# B&R Automation Studio project Soiled_PLC (part 4)

#### pic.st - Implementation code
```iecst
(********************************************************************
 * COPYRIGHT --
 ********************************************************************
 * Program: pic
 * File: pic.st
 * Author: treamsbottom
 * Created: July 16, 2015
 ********************************************************************
 * Implementation of program pic - Pneumatic Incline
 ********************************************************************)
//V1.00.1 First Release
PROGRAM _INIT
//Configuration
mySeq						:= 23;	//Sequence number
myIO						:= 8;
myZone						:= 0;
myRelLine					:= 44;
myBuffBag					:= 0;
myBag						:= 0;
bufferSettleTime			:= 300;
myPI						:= 3;

myOutBag 					:= Line[myRelLine].LastBag;
END_PROGRAM

PROGRAM _CYCLIC
//Inputs

i_bagInIncline			:= X[myIO].X04;
i_cylinderAtBottom		:= X[myIO].X06;
i_cylinderAtTop			:= X[myIO].X05;
i_bagAtBuffer			:= X[myIO].X03;

i_bagAtBufferOut 		:= FALSE; // Any Single bag buffer out IO.
i_bufferOutOpen			:= FALSE;

o_openBuffer			:= FALSE;
o_cylinderDown			:= FALSE;

Request.PI[myPI]		:= FALSE;
RequestRel.PI[myPI]		:= FALSE;

IF (myBag = 0) THEN
//	Alarm[mySeq].Bag	:= mySeq + 10000;
ELSE
//	Alarm[mySeq].Bag	:= myBag;
END_IF;

Alarm[mySeq].Name 		:= 0;
Alarm[mySeq].Bag	:= 10017;
Alarm[mySeq].Beacon	:= TRUE;
Alarm[mySeq].Extra		:= 0;
Alarm[mySeq].Time		:= 3000;

//Setup Sequence
step := D[900 + mySeq];
//Setup Pulse contact
pls := (step <> lastStep);
lastStep := step;

//Sequence
IF (step = 0) THEN
	//Disabled
END_IF;

//Wait for at buffer
ton_10ms_SettledBuffer(IN:= i_bagAtBuffer, PT:= bufferSettleTime);
IF (step = 1) THEN
	IF NOT Std.HaltSysZone[myZone] AND i_cylinderAtTop AND NOT i_bagInIncline THEN
		IF useRequest THEN
			D[900 + mySeq] := 2;
		ELSE
			IF ton_10ms_SettledBuffer.Q THEN
				IF (myBuffBag > 0) THEN
					IF (Bag[myBuffBag].Cat > 0) AND (Bag[myBag].Cat = 0) THEN
						D[900 + mySeq] := 2;
					ELSIF (Bag[myBuffBag].Cat = 0) THEN
						Alarm[mySeq].Name := ALM_BAG_DATA_ERROR;
						Alarm[mySeq].Bag := myBuffBag;
					ELSE
						Alarm[mySeq].Name := ALM_BAG_DATA_ERROR;
					END_IF;
				ELSE
					D[900 + mySeq] := 2;
				END_IF;
			ELSIF (myBuffBag > 0) AND (Bag[myBuffBag].Cat > 0) THEN
				Alarm[mySeq].Name := ALM_BAG_NOT_SETTLED;
			END_IF;
		END_IF;
	ELSIF NOT Std.HaltSysZone[myZone] THEN
		Alarm[mySeq].Name := ALM_SWITCH_FAULT;
	END_IF;
END_IF;

//Open Buffer stop
IF (step = 2) THEN
	releaseValid := ((myBag = 0) OR ((Bag[myBag].Cat = 0) AND (Bag[myBuffBag].Cat > 0)));
	o_openBuffer	   := releaseValid AND NOT useRequest;
	Request.PI[myPI]  := releaseValid AND useRequest;
	IF (i_bagInIncline AND releaseValid) THEN
		IF (myBag > 0) THEN
			Bag[myBag] := Bag[myBuffBag]; //Clear empty buffer bag data if used
			Bag[myBuffBag] := Bag[0];
		END_IF;
		D[900 + mySeq] := 3;
	ELSIF (myBag > 0) THEN
		IF (Bag[myBag].Cat > 0) THEN
			Alarm[mySeq].Name := ALM_BAG_DATA_ERROR;
			Alarm[mySeq].Time := 0;
		ELSIF (Bag[myBuffBag].Cat = 0) THEN
			Alarm[mySeq].Name := ALM_BAG_DATA_ERROR;
			Alarm[mySeq].Bag := myBuffBag;
			Alarm[mySeq].Time := 0;
		ELSE
			Alarm[mySeq].Name  := ALM_BAG_NOT_ARRIVED;
		END_IF;
		Alarm[mySeq].Name  := ALM_BAG_NOT_ARRIVED;
	END_IF;
END_IF;

//Let bag settle at base OF incline
ton_10ms_SettledInIncline(IN:= i_bagInIncline, PT:= 300);
IF (step = 3) THEN
	o_openBuffer := NOT useRequest;
	IF  ton_10ms_SettledInIncline.Q AND NOT Std.HaltSysZone[myZone] THEN
		D[900 + mySeq] := 4;
	ELSIF NOT Std.HaltSysZone[myZone] THEN
		Alarm[mySeq].Name := ALM_BAG_NOT_SETTLED;
	END_IF;
END_IF

//Move incline down to collect first trolley
ton_10ms_CylinderDown(IN := i_cylinderAtBottom, PT:=300);
IF (step = 4) THEN
	o_openBuffer := NOT useRequest;
	o_cylinderDown := TRUE;
	IF ton_10ms_CylinderDown.Q THEN
		D[900 + mySeq] := 5;
	END_IF;
	Alarm[mySeq].Name := ALM_SWITCH_FAULT;
END_IF;

//Let cylinder move back to the top.
IF (step = 5) THEN
	o_openBuffer := NOT useRequest;
	IF i_cylinderAtTop THEN
		D[900 + mySeq] := 6;
	END_IF;
	Alarm[mySeq].Name := ALM_SWITCH_FAULT;
END_IF;

//Check for valid release..
//Check for line space.
IF (step = 6) THEN
	releaseValid := (ton_10ms_SettledInIncline.Q AND NOT i_cylinderAtBottom AND NOT i_bagAtBufferOut AND NOT i_bufferOutOpen AND ((myBag = 0) OR ((Bag[myBag].Cat > 0) AND (Bag[myOutBag].Cat = 0))));
	IF (myRelLine > 0) THEN
		IF (Line[myRelLine].Clear AND releaseValid) THEN
			C[myRelLine] := 0;
			D[900 + mySeq] := 7;
		END_IF;
		IF i_cylinderAtBottom OR NOT i_bagInIncline THEN
			Alarm[mySeq].Name := ALM_SWITCH_FAULT;
			Alarm[mySeq].Time := 0;
		ELSIF (Line[myRelLine].Clear AND i_bagAtBufferOut) THEN
			Alarm[mySeq].Name := ALM_SWITCH_FAULT;
		ELSIF (myBag > 0) AND (Bag[myBag].Cat = 0) THEN
			Alarm[mySeq].Name := ALM_BAG_DATA_ERROR;
			Alarm[mySeq].Time := 0;
		ELSIF Line[myRelLine].Clear AND (myOutBag > 0) AND (Bag[myOutBag].Cat > 0) THEN
			Alarm[mySeq].Name := ALM_BAG_DATA_ERROR;
			Alarm[mySeq].Bag := myOutBag;
			Alarm[mySeq].Time := 0;
		END_IF;
	ELSE
		RequestRel.PI[myPI] := releaseValid;
		IF EnableRel.PI[myPI] AND releaseValid THEN
			D[900 + mySeq] := 7;
		ELSIF NOT i_cylinderAtBottom OR NOT i_bagInIncline THEN
			Alarm[mySeq].Name := ALM_SWITCH_FAULT;
			Alarm[mySeq].Time := 0;
		ELSIF (myBag > 0) AND (Bag[myBag].Cat = 0) THEN
			Alarm[mySeq].Name := ALM_BAG_DATA_ERROR;
			Alarm[mySeq].Time := 0;
		ELSIF (myOutBag > 0) AND (Bag[myOutBag].Cat > 0) THEN
			Alarm[mySeq].Name := ALM_BAG_DATA_ERROR;
			Alarm[mySeq].Bag := myOutBag;
			Alarm[mySeq].Time := 0;
		END_IF;
	END_IF;
END_IF;

//Move cylinder down to get 2nd trolley.
IF (step = 7) THEN
	o_cylinderDown := TRUE;
	IF  ton_10ms_CylinderDown.Q THEN
		D[900 + mySeq] := 8;
	END_IF;
	Alarm[mySeq].Name := ALM_SWITCH_FAULT;
END_IF;

//Release bag
IF (step = 8) THEN
	releaseValid := (NOT i_bagAtBufferOut AND NOT i_bufferOutOpen AND ((myBag = 0) OR ((Bag[myBag].Cat > 0) AND (Bag[myOutBag].Cat = 0))));
	o_cylinderDown := NOT releaseValid; // Hold cylinder down if release is not valid.
	IF releaseValid THEN
		IF (myBag = 0) THEN// Not tracking.
			IF (myRelLine > 0) THEN
				IF Line[myRelLine].Trip THEN
					D[900 + mySeq] := 1;
				END_IF;
			ELSE
				IF NOT EnableRel.PI[myPI] THEN
					D[900 + mySeq] := 1;
				END_IF;
			END_IF;
			IF NOT Std.HaltSysZone[myZone] THEN
				Alarm[mySeq].Name := ALM_BAG_NOT_RELEASED;
			END_IF;
		ELSE//Use tracking
			IF (myRelLine > 0) THEN
				IF Line[myRelLine].Trip THEN
					Bag[myOutBag] := Bag[myBag];
					Bag[myBag] := Bag[0];
					D[900 + mySeq] := 1;
				END_IF;
			ELSE
				IF NOT EnableRel.PI[myPI] AND (Bag[myBag].Cat = 0) THEN // Make sure data is copied out by enabling sequence.
					D[900 + mySeq] := 1;
				ELSIF NOT EnableRel.PI[myPI] AND (Bag[myBag].Cat > 0) THEN
					Alarm[mySeq].Name := ALM_BAG_DATA_ERROR;
				END_IF;
			END_IF;
		END_IF;
	ELSIF i_bagAtBufferOut AND NOT i_bufferOutOpen THEN
		Alarm[mySeq].Name := ALM_SWITCH_FAULT;
		Alarm[mySeq].Time := 0;
	ELSIF (myBag > 0) THEN
		IF (Bag[myBag].Cat = 0) THEN
			Alarm[mySeq].Name := ALM_BAG_DATA_ERROR;
			Alarm[mySeq].Time := 0;
		ELSIF (Bag[myOutBag].Cat > 0) THEN
			Alarm[mySeq].Name := ALM_BAG_DATA_ERROR;
			Alarm[mySeq].Bag := myOutBag;
			Alarm[mySeq].Time := 0;
		END_IF;
	END_IF;
END_IF

//-----------------------------------
//PLC Outputs - adjust TO suit system
//-----------------------------------

Y[11].Y09 := o_cylinderDown;
Y[3].Y15 := o_openBuffer;

//Alarms
timerAlarm(IN := NOT pls AND (Alarm[mySeq].Name > 0),PT:= Alarm[mySeq].Time);

Alarm[mySeq].On 	:= timerAlarm.Q;
Alarm[mySeq].ET 	:= timerAlarm.ET;

END_PROGRAM
```

#### pic.var - Local variables
```iecst
(********************************************************************
 * COPYRIGHT --
 ********************************************************************
 * Program: pr
 * File: pr.var
 * Author: treamsbottom
 * Created: July 16, 2015
 ********************************************************************
 * Local variables of program pr
 ********************************************************************)
VAR
	mySeq : UINT;
	myIO : UINT;
	myZone : UINT;
	myRelLine : UINT;
	myBag : UINT;
	i_bagAtBuffer : BOOL;
	i_bagAtBufferOut : BOOL;
	i_bufferOutOpen : BOOL;
	o_openBuffer : BOOL;
	step : UINT;
	pls : BOOL;
	timerAlarm : TON_10ms;
END_VAR
VAR RETAIN
	lastStep : UINT;
END_VAR
VAR
	bufferSettleTime : UDINT;
	myOutBag : UINT;
	myBuffBag : UINT;
	myPI : UINT;
	i_bagInIncline : BOOL;
	i_cylinderAtBottom : BOOL;
	i_cylinderAtTop : BOOL;
	o_cylinderDown : BOOL;
	useRequest : BOOL;
	releaseValid : BOOL;
	ton_10ms_SettledBuffer : TON_10ms;
	ton_10ms_SettledInIncline : TON_10ms;
	ton_10ms_CylinderDown : TON_10ms;
END_VAR
```

### Program Logical/Sequences/10ms/24_cpi4 (IEC) - *Pneumatic Incline

#### pic.st
```iecst
(********************************************************************
 * COPYRIGHT --
 ********************************************************************
 * Program: pic
 * File: pic.st
 * Author: treamsbottom
 * Created: July 16, 2015
 ********************************************************************
 * Implementation of program pic - Pneumatic Incline
 ********************************************************************)
//V1.00.1 First Release
PROGRAM _INIT
//Configuration
mySeq						:= 24;	//Sequence number
myIO						:= 7;
myZone						:= 0;
myRelLine					:= 41;
myBuffBag					:= 0;
myBag						:= 0;
bufferSettleTime			:= 300;
myPI						:= 4;

myOutBag 					:= Line[myRelLine].LastBag;
END_PROGRAM

PROGRAM _CYCLIC
//Inputs

i_bagInIncline			:= X[9].X16;
i_cylinderAtBottom		:= X[10].X01;
i_cylinderAtTop			:= X[10].X02;
i_bagAtBuffer			:= X[9].X15;

i_bagAtBufferOut 		:= FALSE; // Any Single bag buffer out IO.
i_bufferOutOpen			:= FALSE;

o_openBuffer			:= FALSE;
o_cylinderDown			:= FALSE;

Request.PI[myPI]		:= FALSE;
RequestRel.PI[myPI]		:= FALSE;

IF (myBag = 0) THEN
//	Alarm[mySeq].Bag	:= mySeq + 10000;
ELSE
//	Alarm[mySeq].Bag	:= myBag;
END_IF;

Alarm[mySeq].Name 		:= 0;
Alarm[mySeq].Bag	:= 10018;
Alarm[mySeq].Beacon	:= TRUE;
Alarm[mySeq].Extra		:= 0;
Alarm[mySeq].Time		:= 3000;

//Setup Sequence
step := D[900 + mySeq];
//Setup Pulse contact
pls := (step <> lastStep);
lastStep := step;

//Sequence
IF (step = 0) THEN
	//Disabled
END_IF;

//Wait for at buffer
ton_10ms_SettledBuffer(IN:= i_bagAtBuffer, PT:= bufferSettleTime);
IF (step = 1) THEN
	IF NOT Std.HaltSysZone[myZone] AND i_cylinderAtTop AND NOT i_bagInIncline THEN
		IF useRequest THEN
			D[900 + mySeq] := 2;
		ELSE
			IF ton_10ms_SettledBuffer.Q THEN
				IF (myBuffBag > 0) THEN
					IF (Bag[myBuffBag].Cat > 0) AND (Bag[myBag].Cat = 0) THEN
						D[900 + mySeq] := 2;
					ELSIF (Bag[myBuffBag].Cat = 0) THEN
						Alarm[mySeq].Name := ALM_BAG_DATA_ERROR;
						Alarm[mySeq].Bag := myBuffBag;
					ELSE
						Alarm[mySeq].Name := ALM_BAG_DATA_ERROR;
					END_IF;
				ELSE
					D[900 + mySeq] := 2;
				END_IF;
			ELSIF (myBuffBag > 0) AND (Bag[myBuffBag].Cat > 0) THEN
				Alarm[mySeq].Name := ALM_BAG_NOT_SETTLED;
			END_IF;
		END_IF;
	ELSIF NOT Std.HaltSysZone[myZone] THEN
		Alarm[mySeq].Name := ALM_SWITCH_FAULT;
	END_IF;
END_IF;

//Open Buffer stop
IF (step = 2) THEN
	releaseValid := ((myBag = 0) OR ((Bag[myBag].Cat = 0) AND (Bag[myBuffBag].Cat > 0)));
	o_openBuffer	   := releaseValid AND NOT useRequest;
	Request.PI[myPI]  := releaseValid AND useRequest;
	IF (i_bagInIncline AND releaseValid) THEN
		IF (myBag > 0) THEN
			Bag[myBag] := Bag[myBuffBag]; //Clear empty buffer bag data if used
			Bag[myBuffBag] := Bag[0];
		END_IF;
		D[900 + mySeq] := 3;
	ELSIF (myBag > 0) THEN
		IF (Bag[myBag].Cat > 0) THEN
			Alarm[mySeq].Name := ALM_BAG_DATA_ERROR;
			Alarm[mySeq].Time := 0;
		ELSIF (Bag[myBuffBag].Cat = 0) THEN
			Alarm[mySeq].Name := ALM_BAG_DATA_ERROR;
			Alarm[mySeq].Bag := myBuffBag;
			Alarm[mySeq].Time := 0;
		ELSE
			Alarm[mySeq].Name  := ALM_BAG_NOT_ARRIVED;
		END_IF;
		Alarm[mySeq].Name  := ALM_BAG_NOT_ARRIVED;
	END_IF;
END_IF;

//Let bag settle at base OF incline
ton_10ms_SettledInIncline(IN:= i_bagInIncline, PT:= 300);
IF (step = 3) THEN
	o_openBuffer := NOT useRequest;
	IF  ton_10ms_SettledInIncline.Q AND NOT Std.HaltSysZone[myZone] THEN
		D[900 + mySeq] := 4;
	ELSIF NOT Std.HaltSysZone[myZone] THEN
		Alarm[mySeq].Name := ALM_BAG_NOT_SETTLED;
	END_IF;
END_IF

//Move incline down to collect first trolley
ton_10ms_CylinderDown(IN := i_cylinderAtBottom, PT:=300);
IF (step = 4) THEN
	o_openBuffer := NOT useRequest;
	o_cylinderDown := TRUE;
	IF ton_10ms_CylinderDown.Q THEN
		D[900 + mySeq] := 5;
	END_IF;
	Alarm[mySeq].Name := ALM_SWITCH_FAULT;
END_IF;

//Let cylinder move back to the top.
IF (step = 5) THEN
	o_openBuffer := NOT useRequest;
	IF i_cylinderAtTop THEN
		D[900 + mySeq] := 6;
	END_IF;
	Alarm[mySeq].Name := ALM_SWITCH_FAULT;
END_IF;

//Check for valid release..
//Check for line space.
IF (step = 6) THEN
	releaseValid := ( NOT i_cylinderAtBottom AND NOT i_bagAtBufferOut AND NOT i_bufferOutOpen AND ((myBag = 0) OR ((Bag[myBag].Cat > 0) AND (Bag[myOutBag].Cat = 0))));
	IF (myRelLine > 0) THEN
		IF (Line[myRelLine].Clear AND releaseValid) THEN
			C[myRelLine] := 0;
			D[900 + mySeq] := 7;
		END_IF;
		IF i_cylinderAtBottom OR NOT i_bagInIncline THEN
			Alarm[mySeq].Name := ALM_SWITCH_FAULT;
			Alarm[mySeq].Time := 0;
		ELSIF (Line[myRelLine].Clear AND i_bagAtBufferOut) THEN
			Alarm[mySeq].Name := ALM_SWITCH_FAULT;
		ELSIF (myBag > 0) AND (Bag[myBag].Cat = 0) THEN
			Alarm[mySeq].Name := ALM_BAG_DATA_ERROR;
			Alarm[mySeq].Time := 0;
		ELSIF Line[myRelLine].Clear AND (myOutBag > 0) AND (Bag[myOutBag].Cat > 0) THEN
			Alarm[mySeq].Name := ALM_BAG_DATA_ERROR;
			Alarm[mySeq].Bag := myOutBag;
			Alarm[mySeq].Time := 0;
		END_IF;
	ELSE
		RequestRel.PI[myPI] := releaseValid;
		IF EnableRel.PI[myPI] AND releaseValid THEN
			D[900 + mySeq] := 7;
		ELSIF NOT i_cylinderAtBottom OR NOT i_bagInIncline THEN
			Alarm[mySeq].Name := ALM_SWITCH_FAULT;
			Alarm[mySeq].Time := 0;
		ELSIF (myBag > 0) AND (Bag[myBag].Cat = 0) THEN
			Alarm[mySeq].Name := ALM_BAG_DATA_ERROR;
			Alarm[mySeq].Time := 0;
		ELSIF (myOutBag > 0) AND (Bag[myOutBag].Cat > 0) THEN
			Alarm[mySeq].Name := ALM_BAG_DATA_ERROR;
			Alarm[mySeq].Bag := myOutBag;
			Alarm[mySeq].Time := 0;
		END_IF;
	END_IF;
END_IF;

//Move cylinder down to get 2nd trolley.
IF (step = 7) THEN
	o_cylinderDown := TRUE;
	IF  ton_10ms_CylinderDown.Q THEN
		D[900 + mySeq] := 8;
	END_IF;
	Alarm[mySeq].Name := ALM_SWITCH_FAULT;
END_IF;

//Release bag
IF (step = 8) THEN
	releaseValid := (NOT i_bagAtBufferOut AND NOT i_bufferOutOpen AND ((myBag = 0) OR ((Bag[myBag].Cat > 0) AND (Bag[myOutBag].Cat = 0))));
	o_cylinderDown := NOT releaseValid; // Hold cylinder down if release is not valid.
	IF releaseValid THEN
		IF (myBag = 0) THEN// Not tracking.
			IF (myRelLine > 0) THEN
				IF Line[myRelLine].Trip THEN
					D[900 + mySeq] := 1;
				END_IF;
			ELSE
				IF NOT EnableRel.PI[myPI] THEN
					D[900 + mySeq] := 1;
				END_IF;
			END_IF;
			IF NOT Std.HaltSysZone[myZone] THEN
				Alarm[mySeq].Name := ALM_BAG_NOT_RELEASED;
			END_IF;
		ELSE//Use tracking
			IF (myRelLine > 0) THEN
				IF Line[myRelLine].Trip THEN
					Bag[myOutBag] := Bag[myBag];
					Bag[myBag] := Bag[0];
					D[900 + mySeq] := 1;
				END_IF;
			ELSE
				IF NOT EnableRel.PI[myPI] AND (Bag[myBag].Cat = 0) THEN // Make sure data is copied out by enabling sequence.
					D[900 + mySeq] := 1;
				ELSIF NOT EnableRel.PI[myPI] AND (Bag[myBag].Cat > 0) THEN
					Alarm[mySeq].Name := ALM_BAG_DATA_ERROR;
				END_IF;
			END_IF;
		END_IF;
	ELSIF i_bagAtBufferOut AND NOT i_bufferOutOpen THEN
		Alarm[mySeq].Name := ALM_SWITCH_FAULT;
		Alarm[mySeq].Time := 0;
	ELSIF (myBag > 0) THEN
		IF (Bag[myBag].Cat = 0) THEN
			Alarm[mySeq].Name := ALM_BAG_DATA_ERROR;
			Alarm[mySeq].Time := 0;
		ELSIF (Bag[myOutBag].Cat > 0) THEN
			Alarm[mySeq].Name := ALM_BAG_DATA_ERROR;
			Alarm[mySeq].Bag := myOutBag;
			Alarm[mySeq].Time := 0;
		END_IF;
	END_IF;
END_IF

//-----------------------------------
//PLC Outputs - adjust TO suit system
//-----------------------------------

Y[11].Y16 := o_cylinderDown;
Y[3].Y16 := o_openBuffer;

//Alarms
timerAlarm(IN := NOT pls AND (Alarm[mySeq].Name > 0),PT:= Alarm[mySeq].Time);

Alarm[mySeq].On 	:= timerAlarm.Q;
Alarm[mySeq].ET 	:= timerAlarm.ET;

END_PROGRAM
```

### Program Logical/Sequences/10ms/25_cvc1 (IEC) - * SVC1 Full bag up

#### 7_svc1.var
```iecst
VAR RETAIN
	I_CarrAtTop : BOOL;
	I_CarrAtBottom : BOOL;
	STEP : UINT;
	PLS : BOOL;
	LASTSTEP : UINT;
	O_MoveCarrUp : BOOL;
	O_OpenCarrStop : BOOL;
	O_MoveCarrDown : BOOL;
	I_BagOnCarr : BOOL;
END_VAR
VAR
	SettledBuffer : BOOL;
	SettledBufferET : TIME;
	I_BagAtBuffer : BOOL;
	O_OpenEmptyBuffer : BOOL;
	PastEBagIn : BOOL;
	PastEBagInET : TIME;
	O_MoveCarrDownEBagIn : BOOL;
	BagSettledOnCarr : BOOL;
	BagSettledOnCarrET : TIME;
	EBagSettled : BOOL;
	EBagSettledET : TIME;
	BagSettledBuffET : TIME;
	BagSettledBuff : BOOL;
	I_BagReleased : BOOL;
	O_LLBuffOpen : BOOL;
	I_BagAtLLBuff : BOOL;
	I_BagAtFBuffer : BOOL;
	O_MoveCarrDownEBagOut : BOOL;
	TimerAlarm : TON_10ms;
	I_CarrAtEBagOut : BOOL;
	I_CarrAtEBagIn : BOOL;
	I_BagAtEBuffer : BOOL;
	O_OpenFullBuffer : BOOL;
	HighSpeedDone : BOOL;
	MoveUpCollEmpty : BOOL;
	HighSpeedTime : UDINT;
	TONHighSpeed : TON_10ms;
	mySpeed : ARRAY[0..9] OF UINT;
	HS1 : UINT;
	MoveDownEbagOut : BOOL;
	MoveDownBotStep : BOOL;
	MoveUpTopStep : BOOL;
	MoveDownEBagIn : BOOL;
	HighSpeedDoneET : TIME;
	mySeq : UINT;
	I_Disable : BOOL;
	I_CVC5RailDown : BOOL;
	I_LoadingSequence : BOOL;
	I_UnloadingSequence : BOOL;
	I_UpButton : BOOL;
	O_MoveRailIn : BOOL;
	O_MoveRailOut : BOOL;
	RunOn : BOOL;
	RunOnET : TIME;
	O_OpenCarriageStop : BOOL;
	BufferClear : BOOL;
	CarriageClear : BOOL;
	CarriageClearET : TIME;
	MoveUp : BOOL;
	MoveDown : BOOL;
	CVC5Weight : UINT;
	kev : USINT;
	SVC6RailDown : BOOL;
	SVC7RailDown : BOOL;
	SVC5ValidWeight : BOOL;
	Wgt : BOOL;
	SVC5Alarm : UINT;
	PanelPage : UINT;
	TransPanelPage : UINT;
	PasswordCorrect : USINT;
	F1ChangePage : USINT;
	ESCKey : USINT;
	test : UINT;
	SVC1Raw : DINT;
	I_SVC1RailDown : BOOL;
	I_SVC1RailUp : BOOL;
	SVC1ValidWeight : BOOL;
	SVC2RailDown : BOOL;
	SVC3RailDown : BOOL;
	SVC1Alarm : UINT;
	n : USINT;
	PP45Weight : UINT;
	Pushbutton : BOOL;
	PushbuttonET : TIME;
	I_SafeStopOK : BOOL;
	SafeStop : BOOL;
	SafeStopET : TIME;
	O_IndicatorLamp : BOOL;
	LineSpace : UINT;
	SVC2_OK : BOOL;
	SVC3_OK : BOOL;
	BufferBag : UINT;
	LineSearch : ARRAY[0..20] OF UINT;
	Choice : INT;
	LineValid : BOOL;
	SVC1PanelLamp : BOOL;
	O_SVC1PanelLamp : BOOL;
	SVC1AtWeight : BOOL;
	SVC1Amber : BOOL;
	kevin : UINT;
	SVC1Amber1 : BOOL;
	SVC1Amber2 : BOOL;
	kevintest : BOOL;
	FlashAmberLamp : BOOL;
	SVC1AtWeightET : TIME;
	FlashAmberLampET : TIME;
	WeightValid : BOOL;
	WeightValidET : TIME;
	WeightFault : BOOL;
	WeightFaultET : TIME;
	TEST : UINT;
	myReportStn : UINT;
	I_CarriageAtEmptyIn : BOOL;
	I_CarriageAtSafe : BOOL;
	I_EmptyBagAtBuffer : BOOL;
	BagSettledAtBuffer : BOOL;
	BagSettledAtBufferET : UDINT;
	O_OpenBufferStop : BOOL;
	BagSettledOnCarriage : BOOL;
	BagSettledOnCarriageET : UDINT;
	TimeDelay : BOOL;
	TimeDelayET : UDINT;
	I_CarrAtEmptyBagIn : BOOL;
	I_CarriageAtEmptyBagOut : BOOL;
	I_BagAtEmptyBuffer : BOOL;
	I_BagAtFullBuffer : BOOL;
	I_EmptyBagAtBufferStop : BOOL;
	I_FullBagAtBufferStop : BOOL;
	O_EmptyBagAtBufferStop : BOOL;
	O_FullBagAtBufferStop : BOOL;
	O_OpenEmptyBufferStop : BOOL;
	O_OpenFullBufferStop : BOOL;
	O_MoveCarrDown1 : BOOL;
	O_MoveCarrDown2 : BOOL;
	BufferClearET : UDINT;
	BagAtBuffer : BOOL;
	BagAtBufferET : UDINT;
END_VAR
```

#### 7_svc1Cyclic.ab
```automation-basic
PROGRAM _CYCLIC
	(* cyclic program *)

;--------------------------------------------
;Sequence 7 - SVC1 Vertical conveyor 1 D[907]
;--------------------------------------------

mySeq                   = 25

;Inputs
I_CarrAtTop				= X[3].X15
I_CarrAtBottom			= X[3].X14
I_BagReleased           = X[3].X16
;I_CarriageAtFullBagOut  = X[3].X04

I_BagOnCarr				= X[5].X07
;I_BagAtEmptyBuffer		= X[3].X06
I_BagAtFullBuffer       = X[3].X13 ;bag at full buffer low level

Request.VC[1]           = FALSE
O_OpenEmptyBufferStop	= FALSE ;Y306
O_OpenFullBufferStop    = FALSE ;Y307

O_MoveCarrUp			= FALSE
O_MoveCarrDown			= FALSE
O_MoveCarrDown1         = FALSE
O_MoveCarrDown2         = FALSE
O_OpenCarrStop			= FALSE

Alarm[mySeq].Name 		= 0
Alarm[mySeq].Bag		= 120
Alarm[mySeq].Beacon		= TRUE
Alarm[mySeq].Extra		= 0
Alarm[mySeq].Time		= 6000

;Setup Sequence
STEP = D[900 + mySeq]
;Setup Pulse contact
PLS = (STEP <> LASTSTEP)
LASTSTEP = STEP

;Safety switch check
IF ((STEP = 1) OR (STEP = 8) ) THEN
	IF I_BagOnCarr	OR X[11].X09 THEN
		D[900 + mySeq] = 0
	ENDIF
ENDIF

IF (STEP = 0) AND I_BagOnCarr THEN
	Alarm[mySeq].Time		= 6
	Alarm[mySeq].Name = almCarriageMoveFault
ENDIF

;Sequence
IF (STEP = 0) THEN
	;Disabled
ENDIF

;Move carriage down to empty bag in
IF (STEP = 1) THEN
	O_MoveCarrDown = ( NOT I_CarrAtBottom)
	IF (I_CarrAtBottom  = TRUE) THEN
		D[900 + mySeq] = 2
	ENDIF
	IF NOT Std.EStop THEN
		Alarm[mySeq].Name = ALM_CARRIAGE_MOVE_FAULT
	ENDIF
ENDIF

;full bag at buffer stop
TON_10ms(I_BagAtFullBuffer,200,BagSettledAtBuffer,BagSettledAtBufferET)
IF (STEP = 2) THEN
	IF (NOT I_BagOnCarr AND (BagSettledAtBuffer = TRUE) AND (D[9]>0) AND (Bag[110].Cat>0) AND (Bag[120].Cat = 0)) THEN
		D[900 + mySeq] = 3

	ENDIF
ENDIF

;open buffer stop
IF (STEP = 3) THEN
	O_OpenFullBufferStop = I_CarrAtBottom
	IF I_BagOnCarr THEN
			IF (Bag[110].Cat>0) AND (Bag[120].Cat=0) THEN
			Bag[120] = Bag[110]
			Bag[110] = Bag[0]
		ENDIF
		D[900 + mySeq] = 4
	ENDIF
	Alarm[mySeq].Name = almBagNotArrived
ENDIF

;bag settles on carriage
TON_10ms(I_BagOnCarr,300,BagSettledOnCarr,BagSettledOnCarrET)
IF (STEP = 4) THEN
	IF BagSettledOnCarr THEN

		D[900 + mySeq] = 5
	ENDIF
	Alarm[mySeq].Time		= 1600
	Alarm[mySeq].Name = almBagNotSettled
ENDIF

;move carriage down
IF (STEP = 5) THEN
	O_MoveCarrUp = NOT I_CarrAtTop ;down to empty bag out
	IF I_CarrAtTop AND NOT Enable.VC[1] THEN
		D[900 + mySeq] = 6
	ENDIF
	IF NOT Std.EStop THEN
		Alarm[mySeq].Time		= 1000
		Alarm[mySeq].Name = ALM_CARRIAGE_MOVE_FAULT
	ENDIF
	IF Enable.VC[1] THEN
		Alarm[mySeq].Time		= 10
		Alarm[mySeq].Name = ALM_AIR_PRESSURE_LOW
	ENDIF
	IF X[11].X09 THEN
			D[900 + mySeq] = 0
	ENDIF
ENDIF

;check buffer clear

IF (STEP = 6) THEN
	Request.VC[1] = TRUE
	IF (Enable.VC[1])THEN
		C[22]          = 0
		D[900 + mySeq] = 7
	ENDIF
ENDIF

;Open carr stop
IF (STEP = 7) THEN
	O_OpenCarrStop = I_CarrAtTop
	IF (Line[22].Clear AND NOT I_CarrAtBottom) THEN
		D[900 + mySeq] = 1
	ENDIF
	Alarm[mySeq].Time		= 600
	Alarm[mySeq].Name = ALM_BAG_NOT_RELEASED
ENDIF

;Alarms
TimerAlarm.IN 	= NOT PLS AND (Alarm[mySeq].Name > 0)
TimerAlarm.PT 	= Alarm[mySeq].Time
TimerAlarm FUB TON_10ms()
Alarm[mySeq].On 	= TimerAlarm.Q
Alarm[mySeq].ET 	= TimerAlarm.ET

	;Inverter Speed Selections
	;-------------------------
	;High Speed Used For Up		= 50Hz
;Medium Speed Used For Down	= 50Hz

;Only allow high speed up if starting from the correct position

;PLC Outputs
;-----------
;Outputs

Y[3].Y12 = (O_OpenFullBufferStop AND I_CarrAtBottom)
Y[11].Y01 = (O_MoveCarrUp 	AND NOT I_CarrAtTop)
Y[11].Y02 =  O_MoveCarrDown
Y[11].Y03 = O_OpenCarrStop

;Don't allow forcing of carriage movement and carriage stop
YForceDisable[13].Y01 	= TRUE
YForceDisable[13].Y02 	= TRUE
YForceDisable[13].Y03 	= TRUE
YForceDisable[13].Y04 	= TRUE
END_PROGRAM
```

### Program Logical/Sequences/10ms/26_cp3 (IEC) - * SP2 Empty bags from SDC1/2

#### 12_sp2.var
```iecst
VAR RETAIN
	STEP : UINT;
	PLS : BOOL;
	LASTSTEP : UINT;
END_VAR
VAR
	TimerAlarm : TON_10ms;
	I_BagAtBuffer : ARRAY[0..3] OF BOOL;
	O_OpenBuffer : BOOL;
	SDC2BufferFullET : TIME;
	SDC2BufferFull : BOOL;
	SettledBufferET : TIME;
	SettledBuffer : ARRAY[0..3] OF BOOL;
	O_OpenSP2BufferStop : BOOL;
	O_SelectPoint : BOOL;
	SP2BufferFull : BOOL;
	SP2BufferFullET : UDINT;
	ParingLoopEnabled : BOOL;
	BagInLoopHasDest : BOOL;
	O_OpenSDC1BufferStop : BOOL;
	BagSettledAtBuffer : BOOL;
	BagSettledAtBufferET : UDINT;
	Alternator : USINT;
	I_OnLineA : BOOL;
	I_TiltA : BOOL;
	I_TiltB : BOOL;
	I_Bagout : BOOL;
	O_OpenBufferStop : BOOL;
	O_SelectLineA : BOOL;
	O_SelectLineB : BOOL;
	O_OpenStops : BOOL;
	O_TiltCylinder : BOOL;
	O_OperatePusher : BOOL;
	PointReset : BOOL;
	PointResetET : UDINT;
	BagAtTilt : BOOL;
	BagAtTiltET : UDINT;
	TiltDown : BOOL;
	TiltDownET : UDINT;
	TiltUp : BOOL;
	TiltUpET : UDINT;
	NotFull : BOOL;
	NotFullET : UDINT;
	Pushed : BOOL;
	SBSN1 : BOOL;
	SBSN1ET : UDINT;
	RequirePusherET : UDINT;
	PushedET : UDINT;
	I_BagAtBufferStop : BOOL;
	O_SP7ToSVC1 : BOOL;
	O_SP7ToSIC3 : BOOL;
	SDC1EmptyBufferFull : BOOL;
	SDC1EmptyBufferFullET : UDINT;
	Reset : BOOL;
	ResetET : UDINT;
	ResetPoint : BOOL;
	I_SDC1EmptyBagAtBuffer : BOOL;
	O_ResetPoints : BOOL;
	BagSettledSDC1Buffer : BOOL;
	BagSettledSDC1BufferET : UDINT;
	BagSettledSDC2Buffer : BOOL;
	BagSettledSDC2BufferET : UDINT;
	MySeq : USINT;
	BagSettledBufferET : ARRAY[0..3] OF UDINT;
	Alt : USINT;
	O_SelectCDC4 : BOOL;
	O_SelectStraight : BOOL;
END_VAR
```

#### 12_sp2Cyclic.ab
```automation-basic
PROGRAM _CYCLIC
	(* cyclic program *)

;---------------------------------------
;Sequence 12 - SP2 Single point 2 D[912]
;---------------------------------------

;Inputs

I_BagAtBuffer[1]		= X[4].X14
I_BagAtBuffer[2]		= X[9].X14

MySeq                   = 26

Alarm[MySeq].Name 			= 0
Alarm[MySeq].Bag			= 10019
Alarm[MySeq].Beacon		= TRUE
Alarm[MySeq].Extra			= 0
Alarm[MySeq].Time			= 3000

O_SelectCDC4                = FALSE
O_SelectStraight            = FALSE

;Setup Sequence
STEP = D[900 + MySeq]
;Setup Pulse contact
PLS = (STEP <> LASTSTEP)
LASTSTEP = STEP

;Sequence
;Step 0 - Disabled
IF (STEP = 0) THEN
	;Disabled
ENDIF

;reset points
TON_10ms((STEP = 1),200,Reset,ResetET)
IF (STEP = 1) THEN

	IF (Line[37].Clear) AND NOT Y[3].Y14  THEN
		D[900 + MySeq] = 2
	ENDIF
	ELSE

ENDIF

;check which bag is ready
TON_10ms(I_BagAtBuffer[1],200,SettledBuffer[1],BagSettledBufferET[1])
TON_10ms(I_BagAtBuffer[2],200,SettledBuffer[2],BagSettledBufferET[2])
IF (STEP = 2) THEN
	IF (Line[37].Clear) THEN
		Alt = Alt + 1
		IF (Alt > 2) THEN
			Alt = 0
		ENDIF
		IF SettledBuffer[1] AND (Alt = 1) THEN
			C[37]          = 0
		    D[900 + MySeq] = 3
		ELSE IF SettledBuffer[2] AND (Alt = 2) THEN
			C[37]          = 0
			D[900 + MySeq] = 4
		ENDIF
	ENDIF
ENDIF

;Bag at line
IF (STEP = 3) THEN
	O_SelectCDC4 = TRUE
	IF (Line[37].Trip = TRUE) THEN
		D[900 + MySeq] = 1
	ENDIF
	Alarm[MySeq].Name 	  = almBagNotArrived
ENDIF

;Bag at line
IF (STEP = 4) THEN
	O_SelectStraight = TRUE
	IF (Line[37].Trip = TRUE) THEN
		D[900 + MySeq] = 1
	ENDIF
	Alarm[MySeq].Name 	  = almBagNotArrived
ENDIF

;Alarms
TimerAlarm.IN 	= NOT PLS AND (Alarm[MySeq].Name > 0)
TimerAlarm.PT 	= Alarm[MySeq].Time
TimerAlarm FUB TON_10ms()
Alarm[MySeq].On 	= TimerAlarm.Q
Alarm[MySeq].ET 	= TimerAlarm.ET

;Outputs
Y[4].Y10 = O_SelectCDC4
Y[4].Y11 = O_SelectStraight
END_PROGRAM
```

### Program Logical/Sequences/10ms/27_cp17 (IEC) - * SP2 Empty bags from SDC1/2

#### 12_sp2.var
```iecst
VAR RETAIN
	STEP : UINT;
	PLS : BOOL;
	LASTSTEP : UINT;
END_VAR
VAR
	TimerAlarm : TON_10ms;
	I_BagAtBuffer : ARRAY[0..3] OF BOOL;
	O_OpenBuffer : BOOL;
	SDC2BufferFullET : TIME;
	SDC2BufferFull : BOOL;
	SettledBufferET : TIME;
	SettledBuffer : ARRAY[0..3] OF BOOL;
	O_OpenSP2BufferStop : BOOL;
	O_SelectPoint : BOOL;
	SP2BufferFull : BOOL;
	SP2BufferFullET : UDINT;
	ParingLoopEnabled : BOOL;
	BagInLoopHasDest : BOOL;
	O_OpenSDC1BufferStop : BOOL;
	BagSettledAtBuffer : BOOL;
	BagSettledAtBufferET : UDINT;
	Alternator : USINT;
	I_OnLineA : BOOL;
	I_TiltA : BOOL;
	I_TiltB : BOOL;
	I_Bagout : BOOL;
	O_OpenBufferStop : BOOL;
	O_SelectLineA : BOOL;
	O_SelectLineB : BOOL;
	O_OpenStops : BOOL;
	O_TiltCylinder : BOOL;
	O_OperatePusher : BOOL;
	PointReset : BOOL;
	PointResetET : UDINT;
	BagAtTilt : BOOL;
	BagAtTiltET : UDINT;
	TiltDown : BOOL;
	TiltDownET : UDINT;
	TiltUp : BOOL;
	TiltUpET : UDINT;
	NotFull : BOOL;
	NotFullET : UDINT;
	Pushed : BOOL;
	SBSN1 : BOOL;
	SBSN1ET : UDINT;
	RequirePusherET : UDINT;
	PushedET : UDINT;
	I_BagAtBufferStop : BOOL;
	O_SP7ToSVC1 : BOOL;
	O_SP7ToSIC3 : BOOL;
	SDC1EmptyBufferFull : BOOL;
	SDC1EmptyBufferFullET : UDINT;
	Reset : BOOL;
	ResetET : UDINT;
	ResetPoint : BOOL;
	I_SDC1EmptyBagAtBuffer : BOOL;
	O_ResetPoints : BOOL;
	BagSettledSDC1Buffer : BOOL;
	BagSettledSDC1BufferET : UDINT;
	BagSettledSDC2Buffer : BOOL;
	BagSettledSDC2BufferET : UDINT;
	MySeq : USINT;
	BagSettledBufferET : ARRAY[0..3] OF UDINT;
	Alt : USINT;
	O_SelectCDC4 : BOOL;
	O_SelectStraight : BOOL;
	O_SelectCDC9 : BOOL;
	O_SelectCPI6 : BOOL;
END_VAR
```

#### 12_sp2Cyclic.ab
```automation-basic
PROGRAM _CYCLIC
	(* cyclic program *)

;---------------------------------------
;Sequence 12 - SP2 Single point 2 D[912]
;---------------------------------------

;Inputs

I_BagAtBuffer[1]		= Request.DCEmptyRelease[9]
I_BagAtBuffer[2]		= RequestRel.PI[6]

MySeq                   = 27

Alarm[MySeq].Name 			= 0
Alarm[MySeq].Bag			= 10020
Alarm[MySeq].Beacon		= TRUE
Alarm[MySeq].Extra			= 0
Alarm[MySeq].Time			= 3000

O_SelectCDC9                   = FALSE
O_SelectCPI6                     = FALSE
Enable.DCEmptyRelease[9] = FALSE
EnableRel.PI[6]              = FALSE

;Setup Sequence
STEP = D[900 + MySeq]
;Setup Pulse contact
PLS = (STEP <> LASTSTEP)
LASTSTEP = STEP

;Sequence
;Step 0 - Disabled
IF (STEP = 0) THEN
	;Disabled
ENDIF

;reset points
TON_10ms((STEP = 1),200,Reset,ResetET)
IF (STEP = 1) THEN

	IF (Line[31].Clear)  THEN
		D[900 + MySeq] = 2
	ENDIF
	ELSE

ENDIF

;check which bag is ready
TON_10ms(I_BagAtBuffer[1],200,SettledBuffer[1],BagSettledBufferET[1])
TON_10ms(I_BagAtBuffer[2],200,SettledBuffer[2],BagSettledBufferET[2])
IF (STEP = 2) THEN
	IF (Line[31].Clear) THEN
		Alt = Alt + 1
		IF (Alt > 2) THEN
			Alt = 0
		ENDIF
		IF SettledBuffer[1] AND (Alt = 1) THEN
			C[31]          = 0
		    D[900 + MySeq] = 3
		ELSE IF SettledBuffer[2] AND (Alt = 2) THEN
			C[31]          = 0
			D[900 + MySeq] = 4
		ENDIF
	ENDIF
ENDIF

;Bag at line
IF (STEP = 3) THEN
	O_SelectCDC9   = TRUE
	Enable.DCEmptyRelease[9] = TRUE
	IF (Line[31].Trip = TRUE) THEN
		D[900 + MySeq] = 1
	ENDIF
	Alarm[MySeq].Name 	  = almBagNotArrived
ENDIF

;Bag at line
IF (STEP = 4) THEN
	EnableRel.PI[6] = TRUE
	O_SelectCPI6 = TRUE
	IF (Line[31].Trip = TRUE) THEN
		D[900 + MySeq] = 1
	ENDIF
	Alarm[MySeq].Name 	  = almBagNotArrived
ENDIF

;Alarms
TimerAlarm.IN 	= NOT PLS AND (Alarm[MySeq].Name > 0)
TimerAlarm.PT 	= Alarm[MySeq].Time
TimerAlarm FUB TON_10ms()
Alarm[MySeq].On 	= TimerAlarm.Q
Alarm[MySeq].ET 	= TimerAlarm.ET

;Outputs
Y[2].Y11 = O_SelectCDC9
Y[10].Y13 = O_SelectCPI6
END_PROGRAM
```

### Program Logical/Sequences/10ms/28_cp16 (IEC) - * SP2 Empty bags from SDC1/2

#### 12_sp2.var
```iecst
VAR RETAIN
	STEP : UINT;
	PLS : BOOL;
	LASTSTEP : UINT;
END_VAR
VAR
	TimerAlarm : TON_10ms;
	I_BagAtBuffer : ARRAY[0..3] OF BOOL;
	O_OpenBuffer : BOOL;
	SDC2BufferFullET : TIME;
	SDC2BufferFull : BOOL;
	SettledBufferET : TIME;
	SettledBuffer : ARRAY[0..3] OF BOOL;
	O_OpenSP2BufferStop : BOOL;
	O_SelectPoint : BOOL;
	SP2BufferFull : BOOL;
	SP2BufferFullET : UDINT;
	ParingLoopEnabled : BOOL;
	BagInLoopHasDest : BOOL;
	O_OpenSDC1BufferStop : BOOL;
	BagSettledAtBuffer : BOOL;
	BagSettledAtBufferET : UDINT;
	Alternator : USINT;
	I_OnLineA : BOOL;
	I_TiltA : BOOL;
	I_TiltB : BOOL;
	I_Bagout : BOOL;
	O_OpenBufferStop : BOOL;
	O_SelectLineA : BOOL;
	O_SelectLineB : BOOL;
	O_OpenStops : BOOL;
	O_TiltCylinder : BOOL;
	O_OperatePusher : BOOL;
	PointReset : BOOL;
	PointResetET : UDINT;
	BagAtTilt : BOOL;
	BagAtTiltET : UDINT;
	TiltDown : BOOL;
	TiltDownET : UDINT;
	TiltUp : BOOL;
	TiltUpET : UDINT;
	NotFull : BOOL;
	NotFullET : UDINT;
	Pushed : BOOL;
	SBSN1 : BOOL;
	SBSN1ET : UDINT;
	RequirePusherET : UDINT;
	PushedET : UDINT;
	I_BagAtBufferStop : BOOL;
	O_SP7ToSVC1 : BOOL;
	O_SP7ToSIC3 : BOOL;
	SDC1EmptyBufferFull : BOOL;
	SDC1EmptyBufferFullET : UDINT;
	Reset : BOOL;
	ResetET : UDINT;
	ResetPoint : BOOL;
	I_SDC1EmptyBagAtBuffer : BOOL;
	O_ResetPoints : BOOL;
	BagSettledSDC1Buffer : BOOL;
	BagSettledSDC1BufferET : UDINT;
	BagSettledSDC2Buffer : BOOL;
	BagSettledSDC2BufferET : UDINT;
	MySeq : USINT;
	BagSettledBufferET : ARRAY[0..3] OF UDINT;
	Alt : USINT;
	O_SelectCDC4 : BOOL;
	O_SelectStraight : BOOL;
	O_SelectCDC8 : BOOL;
END_VAR
```

#### 12_sp2Cyclic.ab
```automation-basic
PROGRAM _CYCLIC
	(* cyclic program *)

;---------------------------------------
;Sequence 12 - SP2 Single point 2 D[912]
;---------------------------------------

;Inputs

I_BagAtBuffer[1]		= RequestRel.DC[8]
I_BagAtBuffer[2]		= X[11].X05

MySeq                   = 28

Alarm[MySeq].Name 			= 0
Alarm[MySeq].Bag			= 10021
Alarm[MySeq].Beacon		= TRUE
Alarm[MySeq].Extra			= 0
Alarm[MySeq].Time			= 3000

O_SelectCDC8                    = FALSE
O_SelectStraight                  = FALSE
Enable.DCEmptyRelease[8] = FALSE

;Setup Sequence
STEP = D[900 + MySeq]
;Setup Pulse contact
PLS = (STEP <> LASTSTEP)
LASTSTEP = STEP

;Sequence
;Step 0 - Disabled
IF (STEP = 0) THEN
	;Disabled
ENDIF

;reset points
TON_10ms((STEP = 1),200,Reset,ResetET)
IF (STEP = 1) THEN

	IF Request.PI[6]  THEN
		D[900 + MySeq] = 2
	ENDIF
	ELSE

ENDIF

;check which bag is ready
TON_10ms(I_BagAtBuffer[1],200,SettledBuffer[1],BagSettledBufferET[1])
TON_10ms(I_BagAtBuffer[2],200,SettledBuffer[2],BagSettledBufferET[2])
IF (STEP = 2) THEN
	IF Request.PI[6] THEN
		Alt = Alt + 1
		IF (Alt > 2) THEN
			Alt = 0
		ENDIF
		IF SettledBuffer[1] AND (Alt = 1) THEN
			;C[37]          = 0
		    D[900 + MySeq] = 3
		ELSE IF SettledBuffer[2] AND (Alt = 2) THEN
			;C[37]          = 0
			D[900 + MySeq] = 4
		ENDIF
	ENDIF
ENDIF

;Bag at line
IF (STEP = 3) THEN
	O_SelectCDC8 = TRUE
	Enable.DCEmptyRelease[8] = TRUE
	IF NOT Request.PI[6] THEN
		D[900 + MySeq] = 1
	ENDIF
	Alarm[MySeq].Name 	  = almBagNotArrived
ENDIF

;Bag at line
IF (STEP = 4) THEN
	O_SelectStraight = TRUE
	IF NOT Request.PI[6] THEN
		D[900 + MySeq] = 1
	ENDIF
	Alarm[MySeq].Name 	  = almBagNotArrived
ENDIF

;Alarms
TimerAlarm.IN 	= NOT PLS AND (Alarm[MySeq].Name > 0)
TimerAlarm.PT 	= Alarm[MySeq].Time
TimerAlarm FUB TON_10ms()
Alarm[MySeq].On 	= TimerAlarm.Q
Alarm[MySeq].ET 	= TimerAlarm.ET

;Outputs
;Y[2].Y05 = O_SelectCDC8
Y[10].Y16 = O_SelectStraight
END_PROGRAM
```

### Program Logical/Sequences/10ms/29_cp15 (IEC) - * SP2 Empty bags from SDC1/2

#### 12_sp2.var
```iecst
VAR RETAIN
	STEP : UINT;
	PLS : BOOL;
	LASTSTEP : UINT;
END_VAR
VAR
	TimerAlarm : TON_10ms;
	I_BagAtBuffer : ARRAY[0..3] OF BOOL;
	O_OpenBuffer : BOOL;
	SDC2BufferFullET : TIME;
	SDC2BufferFull : BOOL;
	SettledBufferET : TIME;
	SettledBuffer : ARRAY[0..3] OF BOOL;
	O_OpenSP2BufferStop : BOOL;
	O_SelectPoint : BOOL;
	SP2BufferFull : BOOL;
	SP2BufferFullET : UDINT;
	ParingLoopEnabled : BOOL;
	BagInLoopHasDest : BOOL;
	O_OpenSDC1BufferStop : BOOL;
	BagSettledAtBuffer : BOOL;
	BagSettledAtBufferET : UDINT;
	Alternator : USINT;
	I_OnLineA : BOOL;
	I_TiltA : BOOL;
	I_TiltB : BOOL;
	I_Bagout : BOOL;
	O_OpenBufferStop : BOOL;
	O_SelectLineA : BOOL;
	O_SelectLineB : BOOL;
	O_OpenStops : BOOL;
	O_TiltCylinder : BOOL;
	O_OperatePusher : BOOL;
	PointReset : BOOL;
	PointResetET : UDINT;
	BagAtTilt : BOOL;
	BagAtTiltET : UDINT;
	TiltDown : BOOL;
	TiltDownET : UDINT;
	TiltUp : BOOL;
	TiltUpET : UDINT;
	NotFull : BOOL;
	NotFullET : UDINT;
	Pushed : BOOL;
	SBSN1 : BOOL;
	SBSN1ET : UDINT;
	RequirePusherET : UDINT;
	PushedET : UDINT;
	I_BagAtBufferStop : BOOL;
	O_SP7ToSVC1 : BOOL;
	O_SP7ToSIC3 : BOOL;
	SDC1EmptyBufferFull : BOOL;
	SDC1EmptyBufferFullET : UDINT;
	Reset : BOOL;
	ResetET : UDINT;
	ResetPoint : BOOL;
	I_SDC1EmptyBagAtBuffer : BOOL;
	O_ResetPoints : BOOL;
	BagSettledSDC1Buffer : BOOL;
	BagSettledSDC1BufferET : UDINT;
	BagSettledSDC2Buffer : BOOL;
	BagSettledSDC2BufferET : UDINT;
	MySeq : USINT;
	BagSettledBufferET : ARRAY[0..3] OF UDINT;
	Alt : USINT;
	O_SelectCDC4 : BOOL;
	O_SelectStraight : BOOL;
	O_SelectCDC7 : BOOL;
END_VAR
```

#### 12_sp2Cyclic.ab
```automation-basic
PROGRAM _CYCLIC
	(* cyclic program *)

;---------------------------------------
;Sequence 12 - SP2 Single point 2 D[912]
;---------------------------------------

;Inputs

I_BagAtBuffer[1]		= RequestRel.DC[7]
I_BagAtBuffer[2]		= RequestRel.PI[5]

MySeq                   = 29

Alarm[MySeq].Name 			= 0
Alarm[MySeq].Bag			= 10022
Alarm[MySeq].Beacon		= TRUE
Alarm[MySeq].Extra			= 0
Alarm[MySeq].Time			= 3000

O_SelectCDC7                = FALSE
O_SelectStraight            = FALSE
Enable.DCEmptyRelease[7]    = FALSE
EnableRel.PI[5]             = FALSE

;Setup Sequence
STEP = D[900 + MySeq]
;Setup Pulse contact
PLS = (STEP <> LASTSTEP)
LASTSTEP = STEP

;Sequence
;Step 0 - Disabled
IF (STEP = 0) THEN
	;Disabled
ENDIF

;reset points
TON_10ms((STEP = 1),200,Reset,ResetET)
IF (STEP = 1) THEN

	IF (Line[29].Clear)  THEN
		D[900 + MySeq] = 2
	ENDIF
	ELSE

ENDIF

;check which bag is ready
TON_10ms(I_BagAtBuffer[1],200,SettledBuffer[1],BagSettledBufferET[1])
TON_10ms(I_BagAtBuffer[2],200,SettledBuffer[2],BagSettledBufferET[2])
IF (STEP = 2) THEN
	IF (Line[29].Clear) THEN
		Alt = Alt + 1
		IF (Alt > 2) THEN
			Alt = 0
		ENDIF
		IF SettledBuffer[1] AND (Alt = 1) THEN
			C[29]          = 0
		    D[900 + MySeq] = 3
		ELSE IF SettledBuffer[2] AND (Alt = 2) THEN
			C[29]          = 0
			D[900 + MySeq] = 4
		ENDIF
	ENDIF
ENDIF

;Bag at line
IF (STEP = 3) THEN
	O_SelectCDC7 = TRUE
	Enable.DCEmptyRelease[7] = TRUE
	IF (Line[29].Trip = TRUE) THEN
		D[900 + MySeq] = 1
	ENDIF
	Alarm[MySeq].Name 	  = almBagNotArrived
ENDIF

;Bag at line
IF (STEP = 4) THEN
	EnableRel.PI[5] = TRUE
	O_SelectStraight = TRUE
	IF (Line[29].Trip = TRUE) THEN
		D[900 + MySeq] = 1
	ENDIF
	Alarm[MySeq].Name 	  = almBagNotArrived
ENDIF

;Alarms
TimerAlarm.IN 	= NOT PLS AND (Alarm[MySeq].Name > 0)
TimerAlarm.PT 	= Alarm[MySeq].Time
TimerAlarm FUB TON_10ms()
Alarm[MySeq].On 	= TimerAlarm.Q
Alarm[MySeq].ET 	= TimerAlarm.ET

;Outputs
Y[1].Y15 = O_SelectCDC7
Y[10].Y15 = O_SelectStraight
END_PROGRAM
```

### Program Logical/Sequences/10ms/30_cp14 (IEC) - * SP2 Empty bags from SDC1/2

#### 12_sp2.var
```iecst
VAR RETAIN
	STEP : UINT;
	PLS : BOOL;
	LASTSTEP : UINT;
END_VAR
VAR
	TimerAlarm : TON_10ms;
	I_BagAtBuffer : ARRAY[0..3] OF BOOL;
	O_OpenBuffer : BOOL;
	SDC2BufferFullET : TIME;
	SDC2BufferFull : BOOL;
	SettledBufferET : TIME;
	SettledBuffer : ARRAY[0..3] OF BOOL;
	O_OpenSP2BufferStop : BOOL;
	O_SelectPoint : BOOL;
	SP2BufferFull : BOOL;
	SP2BufferFullET : UDINT;
	ParingLoopEnabled : BOOL;
	BagInLoopHasDest : BOOL;
	O_OpenSDC1BufferStop : BOOL;
	BagSettledAtBuffer : BOOL;
	BagSettledAtBufferET : UDINT;
	Alternator : USINT;
	I_OnLineA : BOOL;
	I_TiltA : BOOL;
	I_TiltB : BOOL;
	I_Bagout : BOOL;
	O_OpenBufferStop : BOOL;
	O_SelectLineA : BOOL;
	O_SelectLineB : BOOL;
	O_OpenStops : BOOL;
	O_TiltCylinder : BOOL;
	O_OperatePusher : BOOL;
	PointReset : BOOL;
	PointResetET : UDINT;
	BagAtTilt : BOOL;
	BagAtTiltET : UDINT;
	TiltDown : BOOL;
	TiltDownET : UDINT;
	TiltUp : BOOL;
	TiltUpET : UDINT;
	NotFull : BOOL;
	NotFullET : UDINT;
	Pushed : BOOL;
	SBSN1 : BOOL;
	SBSN1ET : UDINT;
	RequirePusherET : UDINT;
	PushedET : UDINT;
	I_BagAtBufferStop : BOOL;
	O_SP7ToSVC1 : BOOL;
	O_SP7ToSIC3 : BOOL;
	SDC1EmptyBufferFull : BOOL;
	SDC1EmptyBufferFullET : UDINT;
	Reset : BOOL;
	ResetET : UDINT;
	ResetPoint : BOOL;
	I_SDC1EmptyBagAtBuffer : BOOL;
	O_ResetPoints : BOOL;
	BagSettledSDC1Buffer : BOOL;
	BagSettledSDC1BufferET : UDINT;
	BagSettledSDC2Buffer : BOOL;
	BagSettledSDC2BufferET : UDINT;
	MySeq : USINT;
	BagSettledBufferET : ARRAY[0..3] OF UDINT;
	Alt : USINT;
	O_SelectCDC4 : BOOL;
	O_SelectStraight : BOOL;
	O_SelectCDC6 : BOOL;
END_VAR
```

#### 12_sp2Cyclic.ab
```automation-basic
PROGRAM _CYCLIC
	(* cyclic program *)

;---------------------------------------
;Sequence 12 - SP2 Single point 2 D[912]
;---------------------------------------

;Inputs

I_BagAtBuffer[1]		= RequestRel.DC[6]
I_BagAtBuffer[2]		= X[10].X14

MySeq                   = 30

Alarm[MySeq].Name 			= 0
Alarm[MySeq].Bag			= 10023
Alarm[MySeq].Beacon		= TRUE
Alarm[MySeq].Extra			= 0
Alarm[MySeq].Time			= 3000

O_SelectCDC6                    = FALSE
O_SelectStraight                  = FALSE

Enable.DCEmptyRelease[6] = FALSE

;Setup Sequence
STEP = D[900 + MySeq]
;Setup Pulse contact
PLS = (STEP <> LASTSTEP)
LASTSTEP = STEP

;Sequence
;Step 0 - Disabled
IF (STEP = 0) THEN
	;Disabled
ENDIF

;reset points
TON_10ms((STEP = 1),200,Reset,ResetET)
IF (STEP = 1) THEN

	IF Request.PI[5]  THEN
		D[900 + MySeq] = 2
	ENDIF
	ELSE

ENDIF

;check which bag is ready
TON_10ms(I_BagAtBuffer[1],200,SettledBuffer[1],BagSettledBufferET[1])
TON_10ms(I_BagAtBuffer[2],200,SettledBuffer[2],BagSettledBufferET[2])
IF (STEP = 2) THEN
	IF Request.PI[5] THEN
		Alt = Alt + 1
		IF (Alt > 2) THEN
			Alt = 0
		ENDIF
		IF SettledBuffer[1] AND (Alt = 1) THEN
			;C[37]          = 0
		    D[900 + MySeq] = 3
		ELSE IF SettledBuffer[2] AND (Alt = 2) THEN
			;C[37]          = 0
			D[900 + MySeq] = 4
		ENDIF
	ENDIF
ENDIF

;Bag at line
IF (STEP = 3) THEN
	O_SelectCDC6 = TRUE
	Enable.DCEmptyRelease[6] = TRUE
	IF NOT Request.PI[5] THEN
		D[900 + MySeq] = 1
	ENDIF
	Alarm[MySeq].Name 	  = almBagNotArrived
ENDIF

;Bag at line
IF (STEP = 4) THEN
	O_SelectStraight = TRUE
	IF NOT Request.PI[5] THEN
		D[900 + MySeq] = 1
	ENDIF
	Alarm[MySeq].Name 	  = almBagNotArrived
ENDIF

;Alarms
TimerAlarm.IN 	= NOT PLS AND (Alarm[MySeq].Name > 0)
TimerAlarm.PT 	= Alarm[MySeq].Time
TimerAlarm FUB TON_10ms()
Alarm[MySeq].On 	= TimerAlarm.Q
Alarm[MySeq].ET 	= TimerAlarm.ET

;Outputs
;Y[1].Y09 = O_SelectCDC6
Y[10].Y14 = O_SelectStraight
END_PROGRAM
```

### Program Logical/Sequences/10ms/31_cp2 (IEC) - * SP2 Empty bags from SDC1/2

#### 12_sp2Cyclic.ab
```automation-basic
PROGRAM _CYCLIC
	(* cyclic program *)

;---------------------------------------
;Sequence 12 - SP2 Single point 2 D[912]
;---------------------------------------

;Inputs

I_BagAtBuffer[1]		= X[4].X10
I_BagAtBuffer[2]		= X[9].X14

MySeq                   = 31

Alarm[MySeq].Name 			= 0
Alarm[MySeq].Bag			= 136
Alarm[MySeq].Beacon		= TRUE
Alarm[MySeq].Extra			= 0
Alarm[MySeq].Time			= 3000

O_SelectCDC4                = FALSE
O_SelectStraight            = FALSE

;Setup Sequence
STEP = D[900 + MySeq]
;Setup Pulse contact
PLS = (STEP <> LASTSTEP)
LASTSTEP = STEP

;Sequence
;Step 0 - Disabled
IF (STEP = 0) THEN
	;Disabled
ENDIF

;reset points
TON_10ms(I_BagAtBuffer[1],200,SettledBuffer[1],BagSettledBufferET[1])
IF (STEP = 1) THEN

	IF (D[20]>0) AND SettledBuffer[1] AND (Bag[136].Cat >0)   THEN
		D[900 + MySeq] = 2
	ENDIF
	ELSE

ENDIF

;check which bag is ready

IF (STEP = 2) THEN
		IF (Bag[136].Cat > 0) THEN
			IF (D[3000 + Bag[136].Cat] = 14) THEN
				IF (Bag[136].Dst = 0) THEN
					Bag[136].Dst = 14
				ENDIF
			ENDIF
		ENDIF
	IF (D[20]>0) AND SettledBuffer[1] THEN

		IF (Bag[136].Dst = 14) AND Line[14].Clear AND (Bag[79].Cat = 0) AND (Line[14].Space >0) THEN
			C[14]          = 0
		    D[900 + MySeq] = 3
		ELSE IF  Line[24].Clear AND (Bag[149].Cat = 0)AND (Line[24].Space >0) AND  (Bag[136].Dst <> 14) THEN
			C[24]          = 0
			D[900 + MySeq] = 4
		ENDIF
	ENDIF
ENDIF

;select CDC4
IF (STEP = 3) THEN
	O_SelectCDC4 = TRUE
	IF (Line[14].Trip = TRUE) THEN
		IF (Bag[136].Cat>0) AND (Bag[79].Cat=0) THEN
			Bag[79] = Bag[136]
			Bag[136] = Bag[0]
		ENDIF
		D[900 + MySeq] = 1
	ENDIF
	Alarm[MySeq].Name 	  = almBagNotArrived
ENDIF

;Bag at line
IF (STEP = 4) THEN
	O_SelectStraight = TRUE
	IF (Line[24].Trip = TRUE) THEN
		IF (Bag[136].Cat>0) AND (Bag[149].Cat=0) THEN
			Bag[149] = Bag[136]
			Bag[136] = Bag[0]
		ENDIF
		D[900 + MySeq] = 1
	ENDIF
	Alarm[MySeq].Name 	  = almBagNotArrived
ENDIF

;Alarms
TimerAlarm.IN 	= NOT PLS AND (Alarm[MySeq].Name > 0)
TimerAlarm.PT 	= Alarm[MySeq].Time
TimerAlarm FUB TON_10ms()
Alarm[MySeq].On 	= TimerAlarm.Q
Alarm[MySeq].ET 	= TimerAlarm.ET

;Outputs
Y[4].Y07 = O_SelectCDC4
Y[4].Y08 = O_SelectStraight
Y[4].Y12 = O_SelectCDC4 OR O_SelectStraight
END_PROGRAM
```

### Program Logical/Sequences/10ms/32_cp10 (IEC) - * SP2 Empty bags from SDC1/2

#### 12_sp2Cyclic.ab
```automation-basic
PROGRAM _CYCLIC
	(* cyclic program *)

;---------------------------------------
;Sequence 12 - SP2 Single point 2 D[912]
;---------------------------------------

;Inputs

I_BagAtBuffer[1]		= X[4].X14
I_BagAtBuffer[2]		= X[9].X14

MySeq                   = 26

Alarm[MySeq].Name 			= 0
Alarm[MySeq].Bag			= 10001
Alarm[MySeq].Beacon		= TRUE
Alarm[MySeq].Extra			= 0
Alarm[MySeq].Time			= 3000

O_SelectCDC4                = FALSE
O_SelectStraight            = FALSE

;Setup Sequence
STEP = D[900 + MySeq]
;Setup Pulse contact
PLS = (STEP <> LASTSTEP)
LASTSTEP = STEP

;Sequence
;Step 0 - Disabled
IF (STEP = 0) THEN
	;Disabled
ENDIF

;reset points
TON_10ms((STEP = 1),200,Reset,ResetET)
IF (STEP = 1) THEN

	IF (Line[37].Clear)  THEN
		D[900 + MySeq] = 2
	ENDIF
	ELSE

ENDIF

;check which bag is ready
TON_10ms(I_BagAtBuffer[1],200,SettledBuffer[1],BagSettledBufferET[1])
TON_10ms(I_BagAtBuffer[2],200,SettledBuffer[2],BagSettledBufferET[2])
IF (STEP = 2) THEN
	IF (Line[37].Clear) THEN
		Alt = Alt + 1
		IF (Alt > 2) THEN
			Alt = 0
		ENDIF
		IF SettledBuffer[1] AND (Alt = 1) THEN
			C[37]          = 0
		    D[900 + MySeq] = 3
		ELSE IF SettledBuffer[2] AND (Alt = 2) THEN
			C[37]          = 0
			D[900 + MySeq] = 4
		ENDIF
	ENDIF
ENDIF

;Bag at line
IF (STEP = 3) THEN
	O_SelectCDC4 = TRUE
	IF (Line[37].Trip = TRUE) THEN
		D[900 + MySeq] = 1
	ENDIF
	Alarm[MySeq].Name 	  = almBagNotArrived
ENDIF

;Bag at line
IF (STEP = 4) THEN
	O_SelectStraight = TRUE
	IF (Line[37].Trip = TRUE) THEN
		D[900 + MySeq] = 1
	ENDIF
	Alarm[MySeq].Name 	  = almBagNotArrived
ENDIF

;Alarms
TimerAlarm.IN 	= NOT PLS AND (Alarm[MySeq].Name > 0)
TimerAlarm.PT 	= Alarm[MySeq].Time
TimerAlarm FUB TON_10ms()
Alarm[MySeq].On 	= TimerAlarm.Q
Alarm[MySeq].ET 	= TimerAlarm.ET

;Outputs
Y[4].Y10 = O_SelectCDC4
Y[4].Y11 = O_SelectStraight
END_PROGRAM
```

### Program Logical/Sequences/10ms/34_cpi5 (IEC) - *Pneumatic Incline

#### pic.st
```iecst
(********************************************************************
 * COPYRIGHT --
 ********************************************************************
 * Program: pic
 * File: pic.st
 * Author: treamsbottom
 * Created: July 16, 2015
 ********************************************************************
 * Implementation of program pic - Pneumatic Incline
 ********************************************************************)
//V1.00.1 First Release
PROGRAM _INIT
//Configuration
mySeq						:= 34;	//Sequence number
myIO						:= 7;
myZone						:= 0;
myRelLine					:= 0;
myBuffBag					:= 0;
myBag						:= 0;
bufferSettleTime			:= 300;
myPI						:= 5;
useRequest                  := TRUE;
myOutBag 					:= Line[myRelLine].LastBag;
END_PROGRAM

PROGRAM _CYCLIC
//Inputs

i_bagInIncline			:= X[11].X03;
i_cylinderAtBottom		:= X[11].X02;
i_cylinderAtTop			:= X[11].X01;
i_bagAtBuffer			:= X[10].X14;

i_bagAtBufferOut 		:= FALSE; // Any Single bag buffer out IO.
i_bufferOutOpen			:= FALSE;

o_openBuffer			:= FALSE;
o_cylinderDown			:= FALSE;

Request.PI[myPI]		:= FALSE;
RequestRel.PI[myPI]		:= FALSE;

IF (myBag = 0) THEN
	Alarm[mySeq].Bag	:= 10024;
ELSE
	Alarm[mySeq].Bag	:= 10024;
END_IF;

Alarm[mySeq].Name 		:= 0;
Alarm[mySeq].Beacon	:= TRUE;
Alarm[mySeq].Extra		:= 0;
Alarm[mySeq].Time		:= 3000;

//Setup Sequence
step := D[900 + mySeq];
//Setup Pulse contact
pls := (step <> lastStep);
lastStep := step;

//Sequence
IF (step = 0) THEN
	//Disabled
END_IF;

//Wait for at buffer
ton_10ms_SettledBuffer(IN:= i_bagAtBuffer, PT:= bufferSettleTime);
IF (step = 1) THEN
	IF NOT Std.HaltSysZone[myZone] AND i_cylinderAtTop AND NOT i_bagInIncline THEN
		IF useRequest THEN
			D[900 + mySeq] := 2;
		ELSE
			IF ton_10ms_SettledBuffer.Q THEN
				IF (myBuffBag > 0) THEN
					IF (Bag[myBuffBag].Cat > 0) AND (Bag[myBag].Cat = 0) THEN
						D[900 + mySeq] := 2;
					ELSIF (Bag[myBuffBag].Cat = 0) THEN
						Alarm[mySeq].Name := ALM_BAG_DATA_ERROR;
						Alarm[mySeq].Bag := myBuffBag;
					ELSE
						Alarm[mySeq].Name := ALM_BAG_DATA_ERROR;
					END_IF;
				ELSE
					D[900 + mySeq] := 2;
				END_IF;
			ELSIF (myBuffBag > 0) AND (Bag[myBuffBag].Cat > 0) THEN
				Alarm[mySeq].Name := ALM_BAG_NOT_SETTLED;
			END_IF;
		END_IF;
	ELSIF NOT Std.HaltSysZone[myZone] THEN
		Alarm[mySeq].Name := ALM_SWITCH_FAULT;
	END_IF;
END_IF;

//Open Buffer stop
IF (step = 2) THEN
	releaseValid := ((myBag = 0) OR ((Bag[myBag].Cat = 0) AND (Bag[myBuffBag].Cat > 0)));
	o_openBuffer	   := releaseValid AND NOT useRequest;
	Request.PI[myPI]  := releaseValid AND useRequest;
	IF (i_bagInIncline AND releaseValid) THEN
		IF (myBag > 0) THEN
			Bag[myBag] := Bag[myBuffBag]; //Clear empty buffer bag data if used
			Bag[myBuffBag] := Bag[0];
		END_IF;
		D[900 + mySeq] := 3;
	ELSIF (myBag > 0) THEN
		IF (Bag[myBag].Cat > 0) THEN
			Alarm[mySeq].Name := ALM_BAG_DATA_ERROR;
			Alarm[mySeq].Time := 0;
		ELSIF (Bag[myBuffBag].Cat = 0) THEN
			Alarm[mySeq].Name := ALM_BAG_DATA_ERROR;
			Alarm[mySeq].Bag := myBuffBag;
			Alarm[mySeq].Time := 0;
		ELSE
			Alarm[mySeq].Name  := ALM_BAG_NOT_ARRIVED;
		END_IF;
		Alarm[mySeq].Name  := ALM_BAG_NOT_ARRIVED;
	END_IF;
END_IF;

//Let bag settle at base OF incline
ton_10ms_SettledInIncline(IN:= i_bagInIncline, PT:= 300);
IF (step = 3) THEN
	o_openBuffer := NOT useRequest;
	IF  ton_10ms_SettledInIncline.Q AND NOT Std.HaltSysZone[myZone] THEN
		D[900 + mySeq] := 4;
	ELSIF NOT Std.HaltSysZone[myZone] THEN
		Alarm[mySeq].Name := ALM_BAG_NOT_SETTLED;
	END_IF;
END_IF

//Move incline down to collect first trolley
ton_10ms_CylinderDown(IN := i_cylinderAtBottom, PT:=300);
IF (step = 4) THEN
	o_openBuffer := NOT useRequest;
	o_cylinderDown := TRUE;
	IF ton_10ms_CylinderDown.Q THEN
		D[900 + mySeq] := 5;
	END_IF;
	Alarm[mySeq].Name := ALM_SWITCH_FAULT;
END_IF;

//Let cylinder move back to the top.
IF (step = 5) THEN
	o_openBuffer := NOT useRequest;
	IF i_cylinderAtTop THEN
		D[900 + mySeq] := 6;
	END_IF;
	Alarm[mySeq].Name := ALM_SWITCH_FAULT;
END_IF;

//Check for valid release..
//Check for line space.
IF (step = 6) THEN
	releaseValid := ( NOT i_cylinderAtBottom AND NOT i_bagAtBufferOut AND NOT i_bufferOutOpen AND ((myBag = 0) OR ((Bag[myBag].Cat > 0) AND (Bag[myOutBag].Cat = 0))));
	IF (myRelLine > 0) THEN
		IF (Line[myRelLine].Clear AND releaseValid) THEN
			C[myRelLine] := 0;
			D[900 + mySeq] := 7;
		END_IF;
		IF i_cylinderAtBottom OR NOT i_bagInIncline THEN
			Alarm[mySeq].Name := ALM_SWITCH_FAULT;
			Alarm[mySeq].Time := 0;
		ELSIF (Line[myRelLine].Clear AND i_bagAtBufferOut) THEN
			Alarm[mySeq].Name := ALM_SWITCH_FAULT;
		ELSIF (myBag > 0) AND (Bag[myBag].Cat = 0) THEN
			Alarm[mySeq].Name := ALM_BAG_DATA_ERROR;
			Alarm[mySeq].Time := 0;
		ELSIF Line[myRelLine].Clear AND (myOutBag > 0) AND (Bag[myOutBag].Cat > 0) THEN
			Alarm[mySeq].Name := ALM_BAG_DATA_ERROR;
			Alarm[mySeq].Bag := myOutBag;
			Alarm[mySeq].Time := 0;
		END_IF;
	ELSE
		RequestRel.PI[myPI] := releaseValid;
		IF EnableRel.PI[myPI] AND releaseValid THEN
			D[900 + mySeq] := 7;
		ELSIF NOT i_cylinderAtBottom OR NOT i_bagInIncline THEN
			Alarm[mySeq].Name := ALM_SWITCH_FAULT;
			Alarm[mySeq].Time := 0;
		ELSIF (myBag > 0) AND (Bag[myBag].Cat = 0) THEN
			Alarm[mySeq].Name := ALM_BAG_DATA_ERROR;
			Alarm[mySeq].Time := 0;
		ELSIF (myOutBag > 0) AND (Bag[myOutBag].Cat > 0) THEN
			Alarm[mySeq].Name := ALM_BAG_DATA_ERROR;
			Alarm[mySeq].Bag := myOutBag;
			Alarm[mySeq].Time := 0;
		END_IF;
	END_IF;
END_IF;

//Move cylinder down to get 2nd trolley.
IF (step = 7) THEN
	o_cylinderDown := TRUE;
	IF  ton_10ms_CylinderDown.Q THEN
		D[900 + mySeq] := 8;
	END_IF;
	Alarm[mySeq].Name := ALM_SWITCH_FAULT;
END_IF;

//Release bag
IF (step = 8) THEN
	releaseValid := (NOT i_bagAtBufferOut AND NOT i_bufferOutOpen AND ((myBag = 0) OR ((Bag[myBag].Cat > 0) AND (Bag[myOutBag].Cat = 0))));
	o_cylinderDown := NOT releaseValid; // Hold cylinder down if release is not valid.
	IF releaseValid THEN
		IF (myBag = 0) THEN// Not tracking.
			IF (myRelLine > 0) THEN
				IF Line[myRelLine].Trip THEN
					D[900 + mySeq] := 1;
				END_IF;
			ELSE
				IF NOT EnableRel.PI[myPI] THEN
					D[900 + mySeq] := 1;
				END_IF;
			END_IF;
			IF NOT Std.HaltSysZone[myZone] THEN
				Alarm[mySeq].Name := ALM_BAG_NOT_RELEASED;
			END_IF;
		ELSE//Use tracking
			IF (myRelLine > 0) THEN
				IF Line[myRelLine].Trip THEN
					Bag[myOutBag] := Bag[myBag];
					Bag[myBag] := Bag[0];
					D[900 + mySeq] := 1;
				END_IF;
			ELSE
				IF NOT EnableRel.PI[myPI] AND (Bag[myBag].Cat = 0) THEN // Make sure data is copied out by enabling sequence.
					D[900 + mySeq] := 1;
				ELSIF NOT EnableRel.PI[myPI] AND (Bag[myBag].Cat > 0) THEN
					Alarm[mySeq].Name := ALM_BAG_DATA_ERROR;
				END_IF;
			END_IF;
		END_IF;
	ELSIF i_bagAtBufferOut AND NOT i_bufferOutOpen THEN
		Alarm[mySeq].Name := ALM_SWITCH_FAULT;
		Alarm[mySeq].Time := 0;
	ELSIF (myBag > 0) THEN
		IF (Bag[myBag].Cat = 0) THEN
			Alarm[mySeq].Name := ALM_BAG_DATA_ERROR;
			Alarm[mySeq].Time := 0;
		ELSIF (Bag[myOutBag].Cat > 0) THEN
			Alarm[mySeq].Name := ALM_BAG_DATA_ERROR;
			Alarm[mySeq].Bag := myOutBag;
			Alarm[mySeq].Time := 0;
		END_IF;
	END_IF;
END_IF

//-----------------------------------
//PLC Outputs - adjust TO suit system
//-----------------------------------

Y[8].Y15 := o_cylinderDown;
//Y[10].Y14 := o_openBuffer;

//Alarms
timerAlarm(IN := NOT pls AND (Alarm[mySeq].Name > 0),PT:= Alarm[mySeq].Time);

Alarm[mySeq].On 	:= timerAlarm.Q;
Alarm[mySeq].ET 	:= timerAlarm.ET;

END_PROGRAM
```

### Program Logical/Sequences/10ms/35_cic5 (IEC) - *incline

#### ic.st
```iecst
(********************************************************************
 * COPYRIGHT --
 ********************************************************************
 * Program: ic
 * File: ic.st
 * Author: treamsbottom
 * Created: July 17, 2015
 ********************************************************************
 * Implementation of program Incline conveyor.
 ********************************************************************)
//V1.00.1 First Release
PROGRAM _INIT
//Configuration
mySeq					:= 35;		//Sequence number
myIO					:= 10; 	//Incline Conveyor IO module number
myIC					:= 5;		//Incline Conveyor Number
useRequest				:= FALSE; 	//Use the Request bit. Only use when working with x_1_point. otherwise use RequestRelease as the i_bagAtBuffer.
myBuffBag				:= 153;		//Ingoing Buffer bag number
myBag					:= 152;		//Incline bag number
myRelLine				:= 0;
myOutBag				:= Line[myRelLine].LastBag;	//Outgoing buffer bag number

myZone 					:= 0;
//Timer Values
bufferSettleTime		:= 300;  	// Time for bag to settle at buffer in.
moveUpInclineTime		:= 5;//>>IN SECONDS<< // Time to move bag up incline after closing stop.//Min of 4 to shut buffer stop....

alarm						ACCESS ADR(Alarm[mySeq]);
bag							ACCESS ADR(Bag[myBag]);
bag_buff					ACCESS ADR(Bag[myBuffBag]);
bag_out						ACCESS ADR(Bag[myOutBag]);
line_release				ACCESS ADR(Line[myRelLine]);
END_PROGRAM

PROGRAM _CYCLIC
//Inputs
i_paddleInPosition		:= X[myIO].X08;
i_bagAtBuffer			:= X[myIO].X09;
i_bagInIncline			:= X[myIO].X07;
i_BagReleased			:= FALSE;//X[myIO].X05;  //<--- Bag release trip- only to be used in special cases. Take when using tracked bags, as the next sequence will need to copy data into a transit position

i_bagAtBufferOut 		:= FALSE; // Any Single bag buffer out IO.
i_bufferOutOpen			:= FALSE;

//End of inputs.

o_openBuffer			:= FALSE;
o_runMotor				:= FALSE;

Request.IC[myIC] 		:= FALSE;
RequestRel.IC[myIC] 	:= FALSE;

IF (myBag = 0) THEN
	alarm.Bag	:= 152;
ELSE
	alarm.Bag	:= 152;
END_IF;

alarm.Name 		:= 0;
alarm.Beacon		:= TRUE;
alarm.Extra		:= 0;
alarm.Time		:= 3000;

//Setup Sequence
step := D[900 + mySeq];
//Setup Pulse contact
pls := (step <> laststep);
laststep := step;

//Sequence
IF (step = 0) THEN
	//Disabled
END_IF;

//Run Incline until paddle in position
IF (step = 1) THEN
	o_runMotor := NOT i_paddleInPosition;
	IF i_paddleInPosition THEN
		D[900 + mySeq] := 2;
		Count[mySeq] := Count[mySeq] + 1;
	END_IF;
	IF NOT Std.HaltSysZone[myZone] THEN
		alarm.Name := ALM_SWITCH_FAULT;
	END_IF;
END_IF;

//Wait for at buffer
ton_10ms_SettledBuffer(IN:= i_bagAtBuffer, PT:= bufferSettleTime);
IF (step = 2) THEN
	IF NOT i_bagInIncline THEN
		IF useRequest THEN
			D[900 + mySeq] := 3;
		ELSE
			IF ton_10ms_SettledBuffer.Q THEN
				IF (myBuffBag > 0) THEN
					IF (bag_buff.Cat > 0) AND (bag.Cat = 0) THEN
						D[900 + mySeq] := 3;
					ELSIF (bag_buff.Cat = 0) THEN
						alarm.Name := ALM_BAG_DATA_ERROR;
						alarm.Bag := myBuffBag;
					ELSE
						alarm.Name := ALM_BAG_DATA_ERROR;
					END_IF;
				ELSE
					D[900 + mySeq] := 3;
				END_IF;
			ELSIF (myBuffBag > 0) AND (bag_buff.Cat > 0) THEN
				alarm.Name := ALM_BAG_NOT_SETTLED;
			END_IF;
		END_IF;
	ELSE
		alarm.Name := ALM_SWITCH_FAULT;
	END_IF;
END_IF;

//Open Buffer stop
IF (step = 3) THEN
	releaseValid := ((myBag = 0) OR ((bag.Cat = 0) AND (bag_buff.Cat > 0)));
	o_openBuffer	   := releaseValid AND NOT useRequest;
	Request.IC[myIC]  := releaseValid AND useRequest;
	IF i_bagInIncline AND releaseValid THEN
		IF (myBag > 0) THEN
			bag := bag_buff; //Clear empty buffer bag data if used
			bag_buff := Bag[0];
		END_IF;
		D[900 + mySeq] := 4;
	ELSIF (myBag > 0) THEN
		IF (bag.Cat > 0) THEN
			alarm.Name := ALM_BAG_DATA_ERROR;
			alarm.Time := 0;
		ELSIF (bag_buff.Cat = 0) THEN
			alarm.Name := ALM_BAG_DATA_ERROR;
			alarm.Bag := myBuffBag;
			alarm.Time := 0;
		ELSE
			alarm.Name  := ALM_BAG_NOT_ARRIVED;
		END_IF;
	ELSE
		alarm.Name  := ALM_BAG_NOT_ARRIVED;
	END_IF;
END_IF;

ton_10ms_SettledIncline(IN:= (step = 4), PT:= 300);
IF (step = 4) THEN
	o_openBuffer := NOT useRequest;
	IF ton_10ms_SettledIncline.Q THEN
		D[900 + mySeq] := 5;
	END_IF;
END_IF;

//Move Bag up incline
ctu_moveUpIncline(CU:=(step = 5) AND NOT Std.HaltSysZone[myZone] AND Std.Clock1s, RESET := (step <> 5), PV := moveUpInclineTime);
IF (step = 5) THEN
	o_openBuffer 	:= (ctu_moveUpIncline.CV <= 4) AND NOT useRequest;//Close buffer stop after 3 seconds running..
	o_runMotor 		:= TRUE;
	IF ctu_moveUpIncline.Q THEN
		D[900 + mySeq] := 6;
	ELSIF NOT Std.HaltSysZone[myZone] THEN
		alarm.Name := ALM_SWITCH_FAULT;
	END_IF;

END_IF;

//Check for line space.
IF (step = 6) THEN
	releaseValid := (NOT i_bagAtBufferOut AND NOT i_bufferOutOpen AND NOT i_BagReleased AND ((myBag = 0) OR ((bag.Cat > 0) AND (bag_out.Cat = 0))));
	IF (myRelLine > 0) THEN
		IF (line_release.Clear AND releaseValid) THEN
			C[myRelLine] := 0;
			D[900 + mySeq] := 7;
		END_IF;
		IF (line_release.Clear AND i_bagAtBufferOut) THEN
			alarm.Name := ALM_SWITCH_FAULT;
		ELSIF (myBag > 0) AND (bag.Cat = 0) THEN
			alarm.Name := ALM_BAG_DATA_ERROR;
			alarm.Time := 0;
		ELSIF line_release.Clear AND (myOutBag > 0) AND (bag_out.Cat > 0) THEN
			alarm.Name := ALM_BAG_DATA_ERROR;
			alarm.Bag := myOutBag;
			alarm.Time := 0;
		END_IF;
	ELSE
		RequestRel.IC[myIC] := releaseValid;
		IF EnableRel.IC[myIC] AND releaseValid THEN

			D[900 + mySeq] := 7;
		ELSIF (myBag > 0) AND (bag.Cat = 0) THEN
			alarm.Name := ALM_BAG_DATA_ERROR;
			alarm.Time := 0;
		ELSIF (myOutBag > 0) AND (bag_out.Cat > 0) THEN
			alarm.Name := ALM_BAG_DATA_ERROR;
			alarm.Bag := myOutBag;
			alarm.Time := 0;
		END_IF;
	END_IF;
	IF i_BagReleased THEN
		alarm.Name := ALM_SWITCH_FAULT;
		alarm.Time := 0;
	END_IF;
	releaseValid := 0; //Clear this as we are using it as a latch in line 7
END_IF;

//Run motor to release bag.
IF (step = 7) THEN
	IF (NOT i_bagAtBufferOut AND NOT i_bufferOutOpen AND ((myBag = 0) OR ((bag.Cat > 0) AND (bag_out.Cat = 0)))) THEN
		releaseValid := 1;
	END_IF;
	o_runMotor := releaseValid AND NOT Std.HaltSysZone[myZone];
		IF (Bag[152].Cat>0) AND (Bag[166].Cat = 0) THEN
		Bag[166] := Bag[152];
		Bag[152] := Bag[0];
	END_IF
	IF releaseValid THEN
		IF (myBag = 0) THEN
			IF (myRelLine > 0) THEN
				IF line_release.Trip THEN
					D[900 + mySeq] := 1;
				END_IF;
			ELSE
				IF NOT EnableRel.IC[myIC] OR i_BagReleased THEN
					D[900 + mySeq] := 1;
				END_IF;
			END_IF;
			IF NOT Std.HaltSysZone[myZone] THEN
				alarm.Name := ALM_BAG_NOT_RELEASED;
			END_IF;
		ELSE//Use tracking
			IF (myRelLine > 0) THEN
				IF line_release.Trip THEN
					bag_out := bag;
					bag := Bag[0];
					D[900 + mySeq] := 1;
				END_IF;
			ELSE
				IF (i_BagReleased OR NOT EnableRel.IC[myIC]) AND (bag.Cat = 0)  THEN // Make sure data is copied out by enabling sequence.
					D[900 + mySeq] := 1;
				ELSIF NOT EnableRel.IC[myIC] AND (bag.Cat > 0) THEN
					alarm.Name := ALM_BAG_DATA_ERROR;
				END_IF;
			END_IF;
		END_IF;
	ELSIF i_bagAtBufferOut OR i_bufferOutOpen THEN
			alarm.Name := ALM_SWITCH_FAULT;
			alarm.Time := 0;
	ELSIF (myBag > 0) THEN
		IF (bag.Cat = 0) THEN
			alarm.Name := ALM_BAG_DATA_ERROR;
			alarm.Time := 0;
		ELSIF (bag_out.Cat > 0) THEN
			alarm.Name := ALM_BAG_DATA_ERROR;
			alarm.Bag := myOutBag;
			alarm.Time := 0;
		END_IF;
	END_IF;
END_IF;

//-----------------------------------
//PLC Outputs - adjust TO suit system
//-----------------------------------

Y[8].Y13	:= o_runMotor;
Y[2].Y15 := o_openBuffer;

//Alarms
timerAlarm(IN := NOT pls AND (alarm.Name > 0),PT:= alarm.Time);

alarm.On 	:= timerAlarm.Q;
alarm.ET 	:= timerAlarm.ET;;

END_PROGRAM
```

### Program Logical/Sequences/10ms/36_cic6 (IEC) - *incline

#### ic.var
```iecst
(********************************************************************
 * COPYRIGHT --
 ********************************************************************
 * Program: ic
 * File: ic.var
 * Author: treamsbottom
 * Created: July 17, 2015
 ********************************************************************
 * Local variables of program ic
 ********************************************************************)
VAR
	mySeq : UINT;
	myIO : UINT;
	myIC : UINT;
	useRequest : BOOL;
	bufferSettleTime : UDINT;
	myBuffBag : UINT;
	myBag : UINT;
	myRelLine : UINT;
	myOutBag : UINT;
	myZone : UINT;
	i_paddleInPosition : BOOL;
	i_bagAtBuffer : BOOL;
	i_bagAtBufferOut : BOOL;
	i_bufferOutOpen : BOOL;
	o_openBuffer : BOOL;
	o_runMotor : BOOL;
	step : UINT;
	pls : BOOL;
	ton_10ms_SettledBuffer : TON_10ms;
	timerAlarm : TON_10ms;
END_VAR
VAR RETAIN
	laststep : UINT;
END_VAR
VAR
	i_bagInIncline : BOOL;
	moveUpInclineTime : UINT;
	releaseValid : BOOL;
	ton_10ms_SettledIncline : TON_10ms;
	ctu_moveUpIncline : CTU;
	i_BagReleased : BOOL;
	alarm : REFERENCE TO Alm;
	bag : REFERENCE TO Bag_typ;
	bag_buff : REFERENCE TO Bag_typ;
	bag_out : REFERENCE TO Bag_typ;
	line_release : REFERENCE TO Line_Typ;
END_VAR
```

#### ic.st
```iecst
(********************************************************************
 * COPYRIGHT --
 ********************************************************************
 * Program: ic
 * File: ic.st
 * Author: treamsbottom
 * Created: July 17, 2015
 ********************************************************************
 * Implementation of program Incline conveyor.
 ********************************************************************)
//V1.00.1 First Release
PROGRAM _INIT
//Configuration
mySeq					:= 36;		//Sequence number
myIO					:= 171; 	//Incline Conveyor IO module number
myIC					:= 6;		//Incline Conveyor Number
useRequest				:= FALSE; 	//Use the Request bit. Only use when working with x_1_point. otherwise use RequestRelease as the i_bagAtBuffer.
myBuffBag				:= 151;		//Ingoing Buffer bag number
myBag					:= 157;		//Incline bag number
myRelLine				:= 19;
myOutBag				:= Line[myRelLine].LastBag;	//Outgoing buffer bag number

myZone 					:= 0;
//Timer Values
bufferSettleTime		:= 300;  	// Time for bag to settle at buffer in.
moveUpInclineTime		:= 8;//>>IN SECONDS<< // Time to move bag up incline after closing stop.//Min of 4 to shut buffer stop....

alarm						ACCESS ADR(Alarm[mySeq]);
bag							ACCESS ADR(Bag[myBag]);
bag_buff					ACCESS ADR(Bag[myBuffBag]);
bag_out						ACCESS ADR(Bag[myOutBag]);
line_release				ACCESS ADR(Line[myRelLine]);
END_PROGRAM

PROGRAM _CYCLIC
//Inputs
i_paddleInPosition		:= X[10].X13;
i_bagAtBuffer			:= X[2].X16;
i_bagInIncline			:= X[10].X12;
i_BagReleased			:= FALSE;//X[myIO].X05;  //<--- Bag release trip- only to be used in special cases. Take when using tracked bags, as the next sequence will need to copy data into a transit position

i_bagAtBufferOut 		:= FALSE; // Any Single bag buffer out IO.
i_bufferOutOpen			:= FALSE;

//End of inputs.

o_openBuffer			:= FALSE;
o_runMotor				:= FALSE;

Request.IC[myIC] 		:= FALSE;
RequestRel.IC[myIC] 	:= FALSE;

IF (myBag = 0) THEN
	alarm.Bag	:= 157;
ELSE
	alarm.Bag	:= 157;
END_IF;

alarm.Name 		:= 0;
alarm.Beacon		:= TRUE;
alarm.Extra		:= 0;
alarm.Time		:= 3000;

//Setup Sequence
step := D[900 + mySeq];
//Setup Pulse contact
pls := (step <> laststep);
laststep := step;

//Sequence
IF (step = 0) THEN
	//Disabled
END_IF;

//Run Incline until paddle in position
IF (step = 1) THEN
	o_runMotor := NOT i_paddleInPosition;
	IF i_paddleInPosition THEN
		D[900 + mySeq] := 2;
		Count[mySeq] := Count[mySeq] + 1;
	END_IF;
	IF NOT Std.HaltSysZone[myZone] THEN
		alarm.Name := ALM_SWITCH_FAULT;
	END_IF;
END_IF;

//Wait for at buffer
ton_10ms_SettledBuffer(IN:= i_bagAtBuffer, PT:= bufferSettleTime);
IF (step = 2) THEN
	IF NOT i_bagInIncline THEN
		IF useRequest THEN
			D[900 + mySeq] := 3;
		ELSE
			IF ton_10ms_SettledBuffer.Q THEN
				IF (myBuffBag > 0) THEN
					IF (bag_buff.Cat > 0) AND (bag.Cat = 0) THEN
						D[900 + mySeq] := 3;
					ELSIF (bag_buff.Cat = 0) THEN
						alarm.Name := ALM_BAG_DATA_ERROR;
						alarm.Bag := myBuffBag;
					ELSE
						alarm.Name := ALM_BAG_DATA_ERROR;
					END_IF;
				ELSE
					D[900 + mySeq] := 3;
				END_IF;
			ELSIF (myBuffBag > 0) AND (bag_buff.Cat > 0) THEN
				alarm.Name := ALM_BAG_NOT_SETTLED;
			END_IF;
		END_IF;
	ELSE
		alarm.Name := ALM_SWITCH_FAULT;
	END_IF;
END_IF;

//Open Buffer stop
IF (step = 3) THEN
	releaseValid := ((myBag = 0) OR ((bag.Cat = 0) AND (bag_buff.Cat > 0)));
	o_openBuffer	   := releaseValid AND NOT useRequest;
	Request.IC[myIC]  := releaseValid AND useRequest;
	IF i_bagInIncline AND releaseValid THEN
		IF (myBag > 0) THEN
			bag := bag_buff; //Clear empty buffer bag data if used
			bag_buff := Bag[0];
		END_IF;
		D[900 + mySeq] := 4;
	ELSIF (myBag > 0) THEN
		IF (bag.Cat > 0) THEN
			alarm.Name := ALM_BAG_DATA_ERROR;
			alarm.Time := 0;
		ELSIF (bag_buff.Cat = 0) THEN
			alarm.Name := ALM_BAG_DATA_ERROR;
			alarm.Bag := myBuffBag;
			alarm.Time := 0;
		ELSE
			alarm.Name  := ALM_BAG_NOT_ARRIVED;
		END_IF;
	ELSE
		alarm.Name  := ALM_BAG_NOT_ARRIVED;
	END_IF;
END_IF;

ton_10ms_SettledIncline(IN:= (step = 4), PT:= 300);
IF (step = 4) THEN
	o_openBuffer := NOT useRequest;
	IF ton_10ms_SettledIncline.Q THEN
		D[900 + mySeq] := 5;
	END_IF;
END_IF;

//Move Bag up incline
ctu_moveUpIncline(CU:=(step = 5) AND NOT Std.HaltSysZone[myZone] AND Std.Clock1s, RESET := (step <> 5), PV := moveUpInclineTime);
IF (step = 5) THEN
	o_openBuffer 	:= (ctu_moveUpIncline.CV <= 4) AND NOT useRequest;//Close buffer stop after 3 seconds running..
	o_runMotor 		:= TRUE;
	IF ctu_moveUpIncline.Q THEN
		D[900 + mySeq] := 6;
	ELSIF NOT Std.HaltSysZone[myZone] THEN
		alarm.Name := ALM_SWITCH_FAULT;
	END_IF;

END_IF;

//Check for line space.
IF (step = 6) THEN
	releaseValid := (NOT i_bagAtBufferOut AND NOT i_bufferOutOpen AND NOT i_BagReleased AND ((myBag = 0) OR ((bag.Cat > 0) AND (bag_out.Cat = 0))));
	IF (myRelLine > 0) THEN
		IF (line_release.Clear AND releaseValid) THEN
			C[myRelLine] := 0;
			D[900 + mySeq] := 7;
		END_IF;
		IF (line_release.Clear AND i_bagAtBufferOut) THEN
			alarm.Name := ALM_SWITCH_FAULT;
		ELSIF (myBag > 0) AND (bag.Cat = 0) THEN
			alarm.Name := ALM_BAG_DATA_ERROR;
			alarm.Time := 0;
		ELSIF line_release.Clear AND (myOutBag > 0) AND (bag_out.Cat > 0) THEN
			alarm.Name := ALM_BAG_DATA_ERROR;
			alarm.Bag := myOutBag;
			alarm.Time := 0;
		END_IF;
	ELSE
		RequestRel.IC[myIC] := releaseValid;
		IF EnableRel.IC[myIC] AND releaseValid THEN

			D[900 + mySeq] := 7;
		ELSIF (myBag > 0) AND (bag.Cat = 0) THEN
			alarm.Name := ALM_BAG_DATA_ERROR;
			alarm.Time := 0;
		ELSIF (myOutBag > 0) AND (bag_out.Cat > 0) THEN
			alarm.Name := ALM_BAG_DATA_ERROR;
			alarm.Bag := myOutBag;
			alarm.Time := 0;
		END_IF;
	END_IF;
	IF i_BagReleased THEN
		alarm.Name := ALM_SWITCH_FAULT;
		alarm.Time := 0;
	END_IF;
	releaseValid := 0; //Clear this as we are using it as a latch in line 7
END_IF;

//Run motor to release bag.
IF (step = 7) THEN
	IF (NOT i_bagAtBufferOut AND NOT i_bufferOutOpen AND ((myBag = 0) OR ((bag.Cat > 0) AND (bag_out.Cat = 0)))) THEN
		releaseValid := 1;
	END_IF;
	o_runMotor := releaseValid AND NOT Std.HaltSysZone[myZone];
	IF releaseValid THEN
		IF (myBag = 0) THEN
			IF (myRelLine > 0) THEN
				IF line_release.Trip THEN
					D[900 + mySeq] := 1;
				END_IF;
			ELSE
				IF NOT EnableRel.IC[myIC] OR i_BagReleased THEN
					D[900 + mySeq] := 1;
				END_IF;
			END_IF;
			IF NOT Std.HaltSysZone[myZone] THEN
				alarm.Name := ALM_BAG_NOT_RELEASED;
			END_IF;
		ELSE//Use tracking
			IF (myRelLine > 0) THEN
				IF line_release.Trip THEN
					bag_out := bag;
					bag := Bag[0];
					D[900 + mySeq] := 1;
				END_IF;
			ELSE
				IF (i_BagReleased OR NOT EnableRel.IC[myIC]) AND (bag.Cat = 0)  THEN // Make sure data is copied out by enabling sequence.
					D[900 + mySeq] := 1;
				ELSIF NOT EnableRel.IC[myIC] AND (bag.Cat > 0) THEN
					alarm.Name := ALM_BAG_DATA_ERROR;
				END_IF;
			END_IF;
		END_IF;
	ELSIF i_bagAtBufferOut OR i_bufferOutOpen THEN
			alarm.Name := ALM_SWITCH_FAULT;
			alarm.Time := 0;
	ELSIF (myBag > 0) THEN
		IF (bag.Cat = 0) THEN
			alarm.Name := ALM_BAG_DATA_ERROR;
			alarm.Time := 0;
		ELSIF (bag_out.Cat > 0) THEN
			alarm.Name := ALM_BAG_DATA_ERROR;
			alarm.Bag := myOutBag;
			alarm.Time := 0;
		END_IF;
	END_IF;
END_IF;

//-----------------------------------
//PLC Outputs - adjust TO suit system
//-----------------------------------

Y[8].Y14	:= o_runMotor;
Y[2].Y16 := o_openBuffer;

//Alarms
timerAlarm(IN := NOT pls AND (alarm.Name > 0),PT:= alarm.Time);

alarm.On 	:= timerAlarm.Q;
alarm.ET 	:= timerAlarm.ET;;

END_PROGRAM
```

### Program Logical/Sequences/10ms/37_cpi6 (IEC) - *Pneumatic Incline

#### pic.st
```iecst
(********************************************************************
 * COPYRIGHT --
 ********************************************************************
 * Program: pic
 * File: pic.st
 * Author: treamsbottom
 * Created: July 16, 2015
 ********************************************************************
 * Implementation of program pic - Pneumatic Incline
 ********************************************************************)
//V1.00.1 First Release
PROGRAM _INIT
//Configuration
mySeq						:= 37;	//Sequence number
myIO						:= 7;
myZone						:= 0;
myRelLine					:= 0;
myBuffBag					:= 0;
myBag						:= 0;
bufferSettleTime			:= 300;
myPI						:= 6;

myOutBag 					:= Line[myRelLine].LastBag;
END_PROGRAM

PROGRAM _CYCLIC
//Inputs

i_bagInIncline			:= X[11].X08;
i_cylinderAtBottom		:= X[11].X07;
i_cylinderAtTop			:= X[11].X06;
//i_bagAtBuffer			:= X[9].X15;

i_bagAtBufferOut 		:= FALSE; // Any Single bag buffer out IO.
i_bufferOutOpen			:= FALSE;
useRequest                := TRUE;

o_openBuffer			:= FALSE;
o_cylinderDown			:= FALSE;

Request.PI[myPI]		:= FALSE;
RequestRel.PI[myPI]		:= FALSE;

IF (myBag = 0) THEN
	Alarm[mySeq].Bag	:= 10025;
ELSE
	Alarm[mySeq].Bag	:= 10025;
END_IF;

Alarm[mySeq].Name 		:= 0;
Alarm[mySeq].Beacon	:= TRUE;
Alarm[mySeq].Extra		:= 0;
Alarm[mySeq].Time		:= 3000;

//Setup Sequence
step := D[900 + mySeq];
//Setup Pulse contact
pls := (step <> lastStep);
lastStep := step;

//Sequence
IF (step = 0) THEN
	//Disabled
END_IF;

//Wait for at buffer
ton_10ms_SettledBuffer(IN:= i_bagAtBuffer, PT:= bufferSettleTime);
IF (step = 1) THEN
	IF NOT Std.HaltSysZone[myZone] AND i_cylinderAtTop AND NOT i_bagInIncline THEN
		IF useRequest THEN
			D[900 + mySeq] := 2;
		ELSE
			IF ton_10ms_SettledBuffer.Q THEN
				IF (myBuffBag > 0) THEN
					IF (Bag[myBuffBag].Cat > 0) AND (Bag[myBag].Cat = 0) THEN
						D[900 + mySeq] := 2;
					ELSIF (Bag[myBuffBag].Cat = 0) THEN
						Alarm[mySeq].Name := ALM_BAG_DATA_ERROR;
						Alarm[mySeq].Bag := myBuffBag;
					ELSE
						Alarm[mySeq].Name := ALM_BAG_DATA_ERROR;
					END_IF;
				ELSE
					D[900 + mySeq] := 2;
				END_IF;
			ELSIF (myBuffBag > 0) AND (Bag[myBuffBag].Cat > 0) THEN
				Alarm[mySeq].Name := ALM_BAG_NOT_SETTLED;
			END_IF;
		END_IF;
	ELSIF NOT Std.HaltSysZone[myZone] THEN
		Alarm[mySeq].Name := ALM_SWITCH_FAULT;
	END_IF;
END_IF;

//Open Buffer stop
IF (step = 2) THEN
	releaseValid := ((myBag = 0) OR ((Bag[myBag].Cat = 0) AND (Bag[myBuffBag].Cat > 0)));
	o_openBuffer	   := releaseValid AND NOT useRequest;
	Request.PI[myPI]  := releaseValid AND useRequest;
	IF (i_bagInIncline AND releaseValid) THEN
		IF (myBag > 0) THEN
			Bag[myBag] := Bag[myBuffBag]; //Clear empty buffer bag data if used
			Bag[myBuffBag] := Bag[0];
		END_IF;
		D[900 + mySeq] := 3;
	ELSIF (myBag > 0) THEN
		IF (Bag[myBag].Cat > 0) THEN
			Alarm[mySeq].Name := ALM_BAG_DATA_ERROR;
			Alarm[mySeq].Time := 0;
		ELSIF (Bag[myBuffBag].Cat = 0) THEN
			Alarm[mySeq].Name := ALM_BAG_DATA_ERROR;
			Alarm[mySeq].Bag := myBuffBag;
			Alarm[mySeq].Time := 0;
		ELSE
			Alarm[mySeq].Name  := ALM_BAG_NOT_ARRIVED;
		END_IF;
		Alarm[mySeq].Name  := ALM_BAG_NOT_ARRIVED;
	END_IF;
END_IF;

//Let bag settle at base OF incline
ton_10ms_SettledInIncline(IN:= i_bagInIncline, PT:= 300);
IF (step = 3) THEN
	o_openBuffer := NOT useRequest;
	IF  ton_10ms_SettledInIncline.Q AND NOT Std.HaltSysZone[myZone] THEN
		D[900 + mySeq] := 4;
	ELSIF NOT Std.HaltSysZone[myZone] THEN
		Alarm[mySeq].Name := ALM_BAG_NOT_SETTLED;
	END_IF;
END_IF

//Move incline down to collect first trolley
ton_10ms_CylinderDown(IN := i_cylinderAtBottom, PT:=300);
IF (step = 4) THEN
	o_openBuffer := NOT useRequest;
	o_cylinderDown := TRUE;
	IF ton_10ms_CylinderDown.Q THEN
		D[900 + mySeq] := 5;
	END_IF;
	Alarm[mySeq].Name := ALM_SWITCH_FAULT;
END_IF;

//Let cylinder move back to the top.
IF (step = 5) THEN
	o_openBuffer := NOT useRequest;
	IF i_cylinderAtTop THEN
		D[900 + mySeq] := 6;
	END_IF;
	Alarm[mySeq].Name := ALM_SWITCH_FAULT;
END_IF;

//Check for valid release..
//Check for line space.
IF (step = 6) THEN
	releaseValid := (ton_10ms_SettledInIncline.Q AND NOT i_cylinderAtBottom AND NOT i_bagAtBufferOut AND NOT i_bufferOutOpen AND ((myBag = 0) OR ((Bag[myBag].Cat > 0) AND (Bag[myOutBag].Cat = 0))));
	IF (myRelLine > 0) THEN
		IF (Line[myRelLine].Clear AND releaseValid) THEN
			C[myRelLine] := 0;
			D[900 + mySeq] := 7;
		END_IF;
		IF i_cylinderAtBottom OR NOT i_bagInIncline THEN
			Alarm[mySeq].Name := ALM_SWITCH_FAULT;
			Alarm[mySeq].Time := 0;
		ELSIF (Line[myRelLine].Clear AND i_bagAtBufferOut) THEN
			Alarm[mySeq].Name := ALM_SWITCH_FAULT;
		ELSIF (myBag > 0) AND (Bag[myBag].Cat = 0) THEN
			Alarm[mySeq].Name := ALM_BAG_DATA_ERROR;
			Alarm[mySeq].Time := 0;
		ELSIF Line[myRelLine].Clear AND (myOutBag > 0) AND (Bag[myOutBag].Cat > 0) THEN
			Alarm[mySeq].Name := ALM_BAG_DATA_ERROR;
			Alarm[mySeq].Bag := myOutBag;
			Alarm[mySeq].Time := 0;
		END_IF;
	ELSE
		RequestRel.PI[myPI] := releaseValid;
		IF EnableRel.PI[myPI] AND releaseValid THEN
			D[900 + mySeq] := 7;
		ELSIF NOT i_cylinderAtBottom OR NOT i_bagInIncline THEN
			Alarm[mySeq].Name := ALM_SWITCH_FAULT;
			Alarm[mySeq].Time := 0;
		ELSIF (myBag > 0) AND (Bag[myBag].Cat = 0) THEN
			Alarm[mySeq].Name := ALM_BAG_DATA_ERROR;
			Alarm[mySeq].Time := 0;
		ELSIF (myOutBag > 0) AND (Bag[myOutBag].Cat > 0) THEN
			Alarm[mySeq].Name := ALM_BAG_DATA_ERROR;
			Alarm[mySeq].Bag := myOutBag;
			Alarm[mySeq].Time := 0;
		END_IF;
	END_IF;
END_IF;

//Move cylinder down to get 2nd trolley.
IF (step = 7) THEN
	o_cylinderDown := TRUE;
	IF  ton_10ms_CylinderDown.Q THEN
		D[900 + mySeq] := 8;
	END_IF;
	Alarm[mySeq].Name := ALM_SWITCH_FAULT;
END_IF;

//Release bag
IF (step = 8) THEN
	releaseValid := (NOT i_bagAtBufferOut AND NOT i_bufferOutOpen AND ((myBag = 0) OR ((Bag[myBag].Cat > 0) AND (Bag[myOutBag].Cat = 0))));
	o_cylinderDown := NOT releaseValid; // Hold cylinder down if release is not valid.
	IF releaseValid THEN
		IF (myBag = 0) THEN// Not tracking.
			IF (myRelLine > 0) THEN
				IF Line[myRelLine].Trip THEN
					D[900 + mySeq] := 1;
				END_IF;
			ELSE
				IF NOT EnableRel.PI[myPI] THEN
					D[900 + mySeq] := 1;
				END_IF;
			END_IF;
			IF NOT Std.HaltSysZone[myZone] THEN
				Alarm[mySeq].Name := ALM_BAG_NOT_RELEASED;
			END_IF;
		ELSE//Use tracking
			IF (myRelLine > 0) THEN
				IF Line[myRelLine].Trip THEN
					Bag[myOutBag] := Bag[myBag];
					Bag[myBag] := Bag[0];
					D[900 + mySeq] := 1;
				END_IF;
			ELSE
				IF NOT EnableRel.PI[myPI] AND (Bag[myBag].Cat = 0) THEN // Make sure data is copied out by enabling sequence.
					D[900 + mySeq] := 1;
				ELSIF NOT EnableRel.PI[myPI] AND (Bag[myBag].Cat > 0) THEN
					Alarm[mySeq].Name := ALM_BAG_DATA_ERROR;
				END_IF;
			END_IF;
		END_IF;
	ELSIF i_bagAtBufferOut AND NOT i_bufferOutOpen THEN
		Alarm[mySeq].Name := ALM_SWITCH_FAULT;
		Alarm[mySeq].Time := 0;
	ELSIF (myBag > 0) THEN
		IF (Bag[myBag].Cat = 0) THEN
			Alarm[mySeq].Name := ALM_BAG_DATA_ERROR;
			Alarm[mySeq].Time := 0;
		ELSIF (Bag[myOutBag].Cat > 0) THEN
			Alarm[mySeq].Name := ALM_BAG_DATA_ERROR;
			Alarm[mySeq].Bag := myOutBag;
			Alarm[mySeq].Time := 0;
		END_IF;
	END_IF;
END_IF

//-----------------------------------
//PLC Outputs - adjust TO suit system
//-----------------------------------

Y[8].Y16 := o_cylinderDown;
//Y[3].Y16 := o_openBuffer;

//Alarms
timerAlarm(IN := NOT pls AND (Alarm[mySeq].Name > 0),PT:= Alarm[mySeq].Time);

Alarm[mySeq].On 	:= timerAlarm.Q;
Alarm[mySeq].ET 	:= timerAlarm.ET;

END_PROGRAM
```

### Program Logical/Sequences/10ms/38_cp10 (IEC) - * SP2 Empty bags from SDC1/2

#### 12_sp2.var
```iecst
VAR RETAIN
	STEP : UINT;
	PLS : BOOL;
	LASTSTEP : UINT;
END_VAR
VAR
	TimerAlarm : TON_10ms;
	I_BagAtBuffer : ARRAY[0..3] OF BOOL;
	O_OpenBuffer : BOOL;
	SDC2BufferFullET : TIME;
	SDC2BufferFull : BOOL;
	SettledBufferET : TIME;
	SettledBuffer : ARRAY[0..3] OF BOOL;
	O_OpenSP2BufferStop : BOOL;
	O_SelectPoint : BOOL;
	SP2BufferFull : BOOL;
	SP2BufferFullET : UDINT;
	ParingLoopEnabled : BOOL;
	BagInLoopHasDest : BOOL;
	O_OpenSDC1BufferStop : BOOL;
	BagSettledAtBuffer : BOOL;
	BagSettledAtBufferET : UDINT;
	Alternator : USINT;
	I_OnLineA : BOOL;
	I_TiltA : BOOL;
	I_TiltB : BOOL;
	I_Bagout : BOOL;
	O_OpenBufferStop : BOOL;
	O_SelectLineA : BOOL;
	O_SelectLineB : BOOL;
	O_OpenStops : BOOL;
	O_TiltCylinder : BOOL;
	O_OperatePusher : BOOL;
	PointReset : BOOL;
	PointResetET : UDINT;
	BagAtTilt : BOOL;
	BagAtTiltET : UDINT;
	TiltDown : BOOL;
	TiltDownET : UDINT;
	TiltUp : BOOL;
	TiltUpET : UDINT;
	NotFull : BOOL;
	NotFullET : UDINT;
	Pushed : BOOL;
	SBSN1 : BOOL;
	SBSN1ET : UDINT;
	RequirePusherET : UDINT;
	PushedET : UDINT;
	I_BagAtBufferStop : BOOL;
	O_SP7ToSVC1 : BOOL;
	O_SP7ToSIC3 : BOOL;
	SDC1EmptyBufferFull : BOOL;
	SDC1EmptyBufferFullET : UDINT;
	Reset : BOOL;
	ResetET : UDINT;
	ResetPoint : BOOL;
	I_SDC1EmptyBagAtBuffer : BOOL;
	O_ResetPoints : BOOL;
	BagSettledSDC1Buffer : BOOL;
	BagSettledSDC1BufferET : UDINT;
	BagSettledSDC2Buffer : BOOL;
	BagSettledSDC2BufferET : UDINT;
	MySeq : USINT;
	BagSettledBufferET : ARRAY[0..3] OF UDINT;
	Alt : USINT;
	O_SelectCDC4 : BOOL;
	O_SelectStraight : BOOL;
	O_SelectCIC5 : BOOL;
	O_SelectCDC6 : BOOL;
	O_Reset : BOOL;
	O_SelectCDC5 : BOOL;
END_VAR
```

#### 12_sp2Cyclic.ab
```automation-basic
PROGRAM _CYCLIC
	(* cyclic program *)

;---------------------------------------
;Sequence 12 - SP2 Single point 2 D[912]
;---------------------------------------

;Inputs

I_BagAtBuffer[1]		= X[4].X14
I_BagAtBuffer[2]		= X[9].X14

MySeq                   = 38

Alarm[MySeq].Name 			= 0
Alarm[MySeq].Bag			= 10001
Alarm[MySeq].Beacon		= TRUE
Alarm[MySeq].Extra			= 0
Alarm[MySeq].Time			= 3000

O_SelectCIC5                = FALSE
O_SelectCDC6                = FALSE
O_SelectCDC5                = FALSE
EnableRel.IC[2]             = FALSE
O_Reset                     = FALSE

;Setup Sequence
STEP = D[900 + MySeq]
;Setup Pulse contact
PLS = (STEP <> LASTSTEP)
LASTSTEP = STEP

;Sequence
;Step 0 - Disabled
IF (STEP = 0) THEN
	;Disabled
ENDIF

;reset points
TON_10ms((STEP = 1),200,Reset,ResetET)
IF (STEP = 1) THEN
	O_Reset = TRUE
	IF Reset  THEN
		D[900 + MySeq] = 2
	ENDIF
	ELSE

ENDIF

;check which bag is ready

IF (STEP = 2) THEN
	IF (Bag[154].Dst<15) THEN
		Bag[154].Dst = 0
	ENDIF
	IF (Bag[154].Cat>0) AND (Bag[154].Dst>14) THEN
		IF (Bag[154].Dst = 15) AND Line[15].Clear AND (Bag[82].Cat = 0) THEN
			C[15] = 0
			D[938] = 3
		ELSE IF (Bag[154].Dst = 16) AND Line[16].Clear AND (Bag[87].Cat = 0) THEN
				C[16] = 0
				D[938] = 4
		ELSE IF (Bag[154].Dst = 17) AND Line[25].Clear AND (Bag[153].Cat = 0)AND (Line[17].SpaceBIT>0) THEN
			C[25] = 0
			D[938] = 5
		ELSE IF (Bag[154].Dst = 18) AND Line[25].Clear AND (Bag[153].Cat = 0)AND (Line[18].SpaceBIT>0) THEN
			C[25] = 0
			D[938] = 5
		ELSE IF (Bag[154].Dst = 19) AND Line[25].Clear AND (Bag[153].Cat = 0) AND (Line[19].SpaceBIT>0) THEN
			C[25] = 0
			D[938] = 5
		ENDIF
	ENDIF
	IF (Ldg[3].Search = 0) AND RequestRel.IC[2]  AND (Bag[154].Dst=0) THEN
		Ldg[3].Search = 1
	ENDIF
	IF (Ldg[3].Search = 2) THEN
		IF (Ldg[3].Found = 15) AND Line[15].Clear AND (Bag[82].Cat = 0) THEN
			Bag[154].Dst = USINT(Ldg[3].Found)
			C[15] = 0
			D[938] = 3
		ELSE IF (Ldg[3].Found = 16) AND Line[16].Clear AND (Bag[87].Cat = 0) THEN
			Bag[154].Dst = USINT(Ldg[3].Found)
			C[16] = 0
			D[938] = 4
		ELSE IF (Ldg[3].Found = 17) AND Line[25].Clear AND (Bag[153].Cat = 0)AND (Line[17].SpaceBIT>0) THEN
			Bag[154].Dst = USINT(Ldg[3].Found)
			C[25] = 0
			D[938] = 5
		ELSE IF (Ldg[3].Found = 18) AND Line[25].Clear AND (Bag[153].Cat = 0)AND (Line[18].SpaceBIT>0) THEN
			Bag[154].Dst = USINT(Ldg[3].Found)
			C[25] = 0
			D[938] = 5
		ELSE IF (Ldg[3].Found = 19) AND Line[25].Clear AND (Bag[153].Cat = 0) AND (Line[19].SpaceBIT>0) THEN
			Bag[154].Dst = USINT(Ldg[3].Found)
			C[25] = 0
			D[938] = 5
		ENDIF
	ENDIF
	ELSE
	Ldg[3].Found  = 0
	Ldg[3].Search = 0

ENDIF

;Bag at line
IF (STEP = 3) THEN
	O_SelectCDC5 = TRUE
	EnableRel.IC[2] = TRUE
	IF Line[15].Trip AND (Bag[82].Cat = 0) AND (Bag[154].Cat > 0) THEN
		Bag[82] = Bag[154]
		Bag[154] = Bag[0]
		D[938]  = 1
	ENDIF
	Alarm[MySeq].Bag        = 82
	Alarm[MySeq].Name 	  = almBagNotArrived
ENDIF

;Bag at line
IF (STEP = 4) THEN
	O_SelectCDC6 = TRUE
	EnableRel.IC[2] = TRUE
	IF (Line[16].Trip = TRUE) THEN
		IF (Bag[154].Cat > 0) AND (Bag[87].Cat = 0) THEN
			Bag[87] = Bag[154]
			Bag[154]= Bag[0]
			D[900 + MySeq] = 1
		ENDIF
	ENDIF
	Alarm[MySeq].Bag        = 87
	Alarm[MySeq].Name 	  = almBagNotArrived
ENDIF

IF (STEP = 5) THEN
	O_SelectCIC5 = TRUE
	EnableRel.IC[2] = TRUE
	IF (Line[25].Trip = TRUE) THEN
		IF (Bag[154].Cat > 0) AND (Bag[153].Cat = 0) THEN
			Bag[153] = Bag[154]
			Bag[154]= Bag[0]
			D[900 + MySeq] = 1
		ENDIF
		D[900 + MySeq] = 1
	ENDIF
	Alarm[MySeq].Bag        = 153
	Alarm[MySeq].Name 	  = almBagNotArrived
ENDIF

;Alarms
TimerAlarm.IN 	= NOT PLS AND (Alarm[MySeq].Name > 0)
TimerAlarm.PT 	= Alarm[MySeq].Time
TimerAlarm FUB TON_10ms()
Alarm[MySeq].On 	= TimerAlarm.Q
Alarm[MySeq].ET 	= TimerAlarm.ET

;Outputs
Y[1].Y01 = O_SelectCDC5
Y[1].Y07 = O_SelectCDC6
Y[10].Y01 = O_Reset or O_SelectCIC5
Y[10].Y02 = O_Reset or O_SelectCIC5
END_PROGRAM
```

### Program Logical/Sequences/10ms/39_cpc1 (IEC, version 1.00.2) - *Pneumatic VC

#### pc.st - Implementation code
```iecst
(********************************************************************
 * COPYRIGHT --
 ********************************************************************
 * Program: pr
 * File: pr.st
 * Author: treamsbottom
 * Created: July 16, 2015
 ********************************************************************
 * Implementation of program pr
 ********************************************************************)
//V1.00.1 First Release
PROGRAM _INIT
//Configuration
mySeq						:= 39;		//Sequence number
myIO						:= 6;
myX20IO						:= 6;		// IO for hardwired stops
myPC						:= 1;
myZone						:= 0;
myRelLine					:= 46;
useRequest					:= FALSE; 	//Use the Request bit. Only use when working with x_1_point. otherwise use RequestRelease as the i_bagAtBuffer.
myBuffBag					:= 165; 		//Buffer bag
myBag						:= 156; 	//Buffer Bag
bufferSettleTime			:= 300;

isDecline					:= FALSE; // VC is moving bags down
myOutBag 					:= Line[myRelLine].LastBag;
END_PROGRAM

PROGRAM _CYCLIC
//Inputs
i_carrAtTop					:= X[myIO].X03;
i_carrAtBottom				:= X[myIO].X02;
//i_bagArrive					:= X[myIO].X03;
i_bagOnCarriage				:= X[9].X02;
i_bagAtBuffer				:= X[myIO].X01;

i_bagAtBufferOut 		:= FALSE; // Any Single bag buffer out IO.
i_bufferOutOpen			:= FALSE;

o_openBuffer			:= FALSE;
o_openCarriageStop		:= FALSE;
moveToIncomingPosition	:= FALSE;
moveToOutgoingPosition	:= FALSE;

Request.PC[myPC]		:= FALSE;
RequestRel.PC[myPC]		:= FALSE;

IF (myBag = 0) THEN
	Alarm[mySeq].Bag	:= myBag;
ELSE
	Alarm[mySeq].Bag	:= myBag;
END_IF;

Alarm[mySeq].Name 		:= 0;
Alarm[mySeq].Beacon		:= TRUE;
Alarm[mySeq].Extra		:= 0;
Alarm[mySeq].Time		:= 3000;

//Setup Sequence
step := D[900 + mySeq];
//Setup Pulse contact
pls := (step <> lastStep);
lastStep := step;

//Sequence
IF (step = 0) THEN
	//Disabled
END_IF;

//Step 1 move to bag in position
IF (step = 1) THEN
	moveToIncomingPosition := TRUE;
	IF carrInIncomingPos THEN
		D[900 + mySeq] := 2;
	END_IF
	IF NOT Std.HaltSysZone[myZone] THEN
		Alarm[mySeq].Name := ALM_CARRIAGE_MOVE_FAULT;
	END_IF;
END_IF;

//Wait for at buffer
ton_10ms_SettledBuffer(IN:= i_bagAtBuffer, PT:= bufferSettleTime);
IF (step = 2) THEN
	moveToIncomingPosition := TRUE;
	IF carrInIncomingPos AND NOT Std.HaltSysZone[myZone] AND NOT i_bagOnCarriage AND NOT i_bagArrive THEN
		IF useRequest THEN
			D[900 + mySeq] := 3;
		ELSE
			IF ton_10ms_SettledBuffer.Q THEN
				IF (myBuffBag > 0) THEN
					IF (Bag[myBuffBag].Cat > 0) AND (Bag[myBag].Cat = 0) THEN
						D[900 + mySeq] := 3;
					ELSIF (Bag[myBuffBag].Cat = 0) THEN
						Alarm[mySeq].Name := ALM_BAG_DATA_ERROR;
						Alarm[mySeq].Bag := myBuffBag;
					ELSE
						Alarm[mySeq].Name := ALM_BAG_DATA_ERROR;
					END_IF;
				ELSE
					D[900 + mySeq] := 3;
				END_IF;
			ELSIF (myBuffBag > 0) AND (Bag[myBuffBag].Cat > 0) THEN
				Alarm[mySeq].Name := ALM_BAG_NOT_SETTLED;
			END_IF;
		END_IF;
	ELSIF NOT Std.HaltSysZone[myZone] THEN
		Alarm[mySeq].Name := ALM_SWITCH_FAULT;
	END_IF;
	IF 	i_bagOnCarriage THEN
		Alarm[mySeq].Time		:= 300;
		Alarm[mySeq].Name := ALM_SWITCH_FAULT;
	END_IF
END_IF;

//Open Buffer stop
IF (step = 3) THEN
	moveToIncomingPosition := TRUE;
	IF carrInIncomingPos THEN
		carrInPosLatch := TRUE;
	END_IF;
	releaseValid := (carrInPosLatch AND ((myBag = 0) OR ((Bag[myBag].Cat = 0) AND (Bag[myBuffBag].Cat > 0))));
	o_openBuffer	   := releaseValid AND NOT useRequest;
	Request.PC[myPC]  := releaseValid AND useRequest;
	IF ((i_bagArrive OR i_bagOnCarriage) AND releaseValid) THEN
		IF (myBag > 0) THEN
			Bag[myBag] := Bag[myBuffBag]; //Clear empty buffer bag data if used
			Bag[myBuffBag] := Bag[0];
		END_IF;
		D[900 + mySeq] := 4;
	ELSIF (myBag > 0) THEN
		IF (Bag[myBag].Cat > 0) THEN
			Alarm[mySeq].Name := ALM_BAG_DATA_ERROR;
			Alarm[mySeq].Time := 0;
		ELSIF (Bag[myBuffBag].Cat = 0) THEN
			Alarm[mySeq].Name := ALM_BAG_DATA_ERROR;
			Alarm[mySeq].Bag := myBuffBag;
			Alarm[mySeq].Time := 0;
		ELSE
			Alarm[mySeq].Name  := ALM_BAG_NOT_ARRIVED;
		END_IF;
	ELSIF NOT carrInPosLatch THEN
		Alarm[mySeq].Name  := ALM_SWITCH_FAULT;
	ELSE
		Alarm[mySeq].Bag := 165;
		Alarm[mySeq].Time		:= 1000;
		Alarm[mySeq].Name  := ALM_BAG_NOT_ARRIVED;
	END_IF;
END_IF;

// Step 4 Bag settles on carriage..
ton_10ms_SettledCarriage(IN:= i_bagOnCarriage, PT:= 300);
IF (step = 4) THEN
	moveToIncomingPosition := TRUE;
	IF  ton_10ms_SettledCarriage.Q AND NOT Std.HaltSysZone[myZone] AND NOT i_bagArrive THEN
		D[900 + mySeq] := 5;
	ELSIF NOT Std.HaltSysZone[myZone] THEN
		Alarm[mySeq].Name := ALM_BAG_NOT_SETTLED;
	END_IF;
END_IF

// Step 5 move to outgoing position
IF (step = 5) THEN
	moveToOutgoingPosition := TRUE;
	IF carrAtOutgoingPos AND NOT EnableRel.PC[2] THEN
		D[900 + mySeq] := 6;
	ELSIF NOT Std.HaltSysZone[myZone] THEN
		Alarm[mySeq].Name := ALM_CARRIAGE_MOVE_FAULT;
	END_IF;
END_IF;

//Step 6 check release condtion.
//Check for line space.
IF (step = 6) THEN
	moveToOutgoingPosition := TRUE;
	releaseValid := (carrAtOutgoingPos AND ((Bag[myBag].Cat > 0) AND (Bag[myOutBag].Cat = 0)));
	RequestRel.PC[1] := releaseValid ;
	IF EnableRel.PC[2] THEN

			C[46] := 0;
			D[900 + mySeq] := 7;
		//END_IF;
		IF NOT carrAtOutgoingPos THEN
			Alarm[mySeq].Name := ALM_CARRIAGE_MOVE_FAULT;
			Alarm[mySeq].Time := 0;
		ELSIF (Line[myRelLine].Clear AND i_bagAtBufferOut) THEN
			Alarm[mySeq].Name := ALM_SWITCH_FAULT;
		ELSIF (myBag > 0) AND (Bag[myBag].Cat = 0) THEN
			Alarm[mySeq].Name := ALM_BAG_DATA_ERROR;
			Alarm[mySeq].Time := 0;
		ELSIF Line[myRelLine].Clear AND (myOutBag > 0) AND (Bag[myOutBag].Cat > 0) THEN
			Alarm[mySeq].Name := ALM_BAG_DATA_ERROR;
			Alarm[mySeq].Bag := myOutBag;
			Alarm[mySeq].Time := 0;
		END_IF;
	ELSE
		RequestRel.PC[myPC] := releaseValid;
		IF EnableRel.PC[myPC] AND releaseValid THEN
			D[900 + mySeq] := 7;
		ELSIF NOT carrAtOutgoingPos THEN
			Alarm[mySeq].Name := ALM_CARRIAGE_MOVE_FAULT;
			Alarm[mySeq].Time := 0;
		ELSIF (myBag > 0) AND (Bag[myBag].Cat = 0) THEN
			Alarm[mySeq].Name := ALM_BAG_DATA_ERROR;
			Alarm[mySeq].Time := 0;
		ELSIF (myOutBag > 0) AND (Bag[myOutBag].Cat > 0) THEN
			Alarm[mySeq].Name := ALM_BAG_DATA_ERROR;
			Alarm[mySeq].Bag := myOutBag;
			Alarm[mySeq].Time := 0;
		END_IF;
	END_IF;
END_IF;

//Step 7 Release bag.
IF (step = 7) THEN
	releaseValid := i_carrAtTop;
	o_openCarriageStop := i_carrAtTop AND NOT Std.HaltSysZone[myZone];

		IF releaseValid THEN
		IF (myBag = 0) THEN
			IF (myRelLine > 0) THEN
				IF Line[myRelLine].Clear AND NOT i_bagOnCarriage THEN
					D[900 + mySeq] := 1;
				END_IF;
			ELSE
				IF NOT EnableRel.PC[myPC] THEN
					D[900 + mySeq] := 1;
				END_IF;
			END_IF;
			IF NOT Std.HaltSysZone[myZone] THEN
				Alarm[mySeq].Name := ALM_BAG_NOT_RELEASED;
			END_IF;
		ELSE//Use tracking
			IF (myRelLine > 0) THEN
				IF Line[myRelLine].Clear AND NOT i_bagOnCarriage THEN
					Bag[myOutBag] := Bag[myBag];
					Bag[myBag] := Bag[0];
					D[900 + mySeq] := 1;
				ELSIF  i_bagOnCarriage THEN
					Alarm[mySeq].Name := ALM_SWITCH_FAULT;
					Alarm[mySeq].Bag := myBag;
					Alarm[mySeq].Time := 0;
				END_IF;
			ELSE
				IF NOT EnableRel.PC[myPC] AND (Bag[myBag].Cat = 0) THEN // Make sure data is copied out by enabling sequence.
					D[900 + mySeq] := 1;
				ELSIF NOT EnableRel.PC[myPC] AND (Bag[myBag].Cat > 0) THEN
					Alarm[mySeq].Name := ALM_BAG_DATA_ERROR;
				END_IF;
			END_IF;
		END_IF;
	ELSIF NOT carrAtOutgoingPos THEN
		Alarm[mySeq].Name := ALM_CARRIAGE_MOVE_FAULT;
		Alarm[mySeq].Time := 0;
	ELSIF i_bagAtBufferOut AND NOT i_bufferOutOpen THEN
		Alarm[mySeq].Name := ALM_SWITCH_FAULT;
		Alarm[mySeq].Time := 0;
	ELSIF (myBag > 0) THEN
		IF (Bag[myBag].Cat = 0) THEN
			Alarm[mySeq].Name := ALM_BAG_DATA_ERROR;
			Alarm[mySeq].Time := 0;
		ELSIF (Bag[myOutBag].Cat > 0) THEN
			Alarm[mySeq].Name := ALM_BAG_DATA_ERROR;
			Alarm[mySeq].Bag := myOutBag;
			Alarm[mySeq].Time := 0;

		END_IF;
	END_IF;
END_IF;

//Control Position
IF isDecline THEN
	o_moveUp := moveToIncomingPosition;
	o_moveDown := moveToOutgoingPosition;
	carrInIncomingPos := i_carrAtTop;
	carrAtOutgoingPos := i_carrAtBottom;
ELSE
	o_moveDown := moveToIncomingPosition;
	o_moveUp := moveToOutgoingPosition;
	carrInIncomingPos := i_carrAtBottom;
	carrAtOutgoingPos := i_carrAtTop;
END_IF;

//-----------------------------------
//PLC Outputs - adjust TO suit system
//-----------------------------------

Y[5].Y11			:= o_openBuffer;
//Y[myIO].Y07			:= ((step >= 3) AND (step <= 4) AND carrInIncomingPos); //Safe stop

Y[11].Y10 		:= (o_moveUp AND NOT i_carrAtTop); //Move carriage up
Y[11].Y11 		:= (o_moveDown  AND NOT i_carrAtBottom);//Move carriage down
Y[11].Y12 		:= (o_openCarriageStop AND carrAtOutgoingPos);// Carriage Stop

//Don't allow forcing of carriage movement and carriage stop
YForceDisable[myX20IO].Y01 	:= TRUE;
YForceDisable[myX20IO].Y02 	:= TRUE;
YForceDisable[myX20IO].Y03 	:= TRUE;

//Alarms
timerAlarm(IN := NOT pls AND (Alarm[mySeq].Name > 0),PT:= Alarm[mySeq].Time);

Alarm[mySeq].On 	:= timerAlarm.Q;
Alarm[mySeq].ET 	:= timerAlarm.ET;

END_PROGRAM
```

#### pc.var - Local variables
```iecst
(********************************************************************
 * COPYRIGHT --
 ********************************************************************
 * Program: pr
 * File: pr.var
 * Author: treamsbottom
 * Created: July 16, 2015
 ********************************************************************
 * Local variables of program pr
 ********************************************************************)
VAR
	mySeq : UINT;
	myIO : UINT;
	myZone : UINT;
	myRelLine : UINT;
	myBag : UINT;
	i_bagAtBuffer : BOOL;
	i_bagAtBufferOut : BOOL;
	i_bufferOutOpen : BOOL;
	o_openBuffer : BOOL;
	step : UINT;
	pls : BOOL;
	timerAlarm : TON_10ms;
END_VAR
VAR RETAIN
	lastStep : UINT;
END_VAR
VAR
	bufferSettleTime : UDINT;
	myOutBag : UINT;
	myBuffBag : UINT;
	isDecline : BOOL;
	i_carrAtTop : BOOL;
	i_carrAtBottom : BOOL;
	i_bagArrive : BOOL;
	i_bagOnCarriage : BOOL;
	o_moveDown : BOOL;
	o_moveUp : BOOL;
	myPC : UINT;
	useRequest : BOOL;
	o_openCarriageStop : BOOL;
	myX20IO : UINT;
	moveToIncomingPosition : BOOL;
	carrInIncomingPos : BOOL;
	releaseValid : BOOL;
	ton_10ms_SettledBuffer : TON_10ms;
	moveToOutgoingPosition : BOOL;
	carrAtOutgoingPos : BOOL;
	carrInPosLatch : BOOL;
	ton_10ms_SettledCarriage : TON_10ms;
END_VAR
```

### Program Logical/Sequences/10ms/40_cp4 (IEC, version 1.00.0) - * SP2 Empty bags from SDC1/2
